KUKA KRL program: MyProgram_254().src

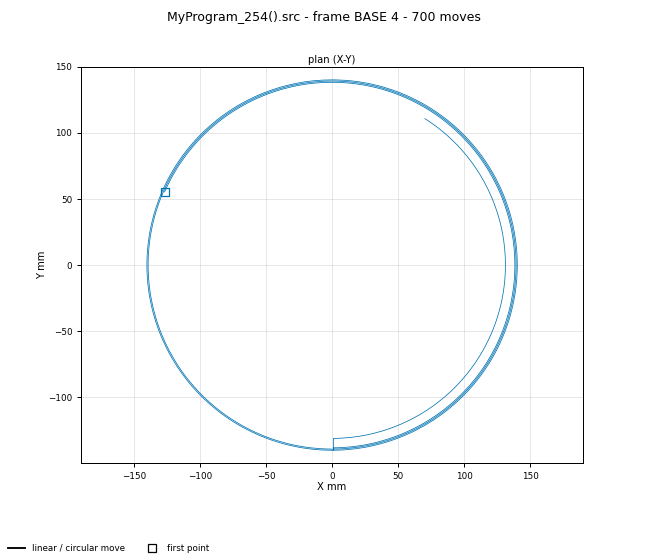
[picture p0: tool path of MyProgram_254().src in frame BASE 4, 700 of 700 moves have a stored position in this frame; points joined in program order, loops and branches not executed]
&ACCESS RVP
&REL 1
&PARAM TEMPLATE = C:\KRC\Roboter\Template\vorgabe
&PARAM EDITMASK = *
DEF MyProgram_254()
; ---- Setting reference (Base) ----
$BASE = BASE_DATA[4]

; --------------------------
; ---- Setting tool (TCP) ----
$TOOL = TOOL_DATA[3]
; --------------------------

$VEL.CP = VEL_APROX_PRINT
Startdeposition()
$VEL.CP = VEL_PRINT
LIN {X -126.8422,Y 55.3756,Z 165,A 156.6903,B 11.101,C 0.1194,E1 10.9554,E2 294.2461} C_DIS
LIN {X -125.3357,Y 58.7076,Z 165,A 155.0353,B 11.101,C 0.1183,E1 10.9574,E2 295.9168} C_DIS
LIN {X -122.9078,Y 63.6351,Z 165,A 152.7935,B 11.1012,C 0.1116,E1 10.9602,E2 298.152} C_DIS
LIN {X -120.9486,Y 67.2845,Z 165,A 151.0182,B 11.1012,C 0.1084,E1 10.9626,E2 299.9329} C_DIS
LIN {X -118.7949,Y 71.0176,Z 165,A 149.2267,B 11.1012,C 0.104,E1 10.9651,E2 301.7233} C_DIS
LIN {X -116.5286,Y 74.6779,Z 165,A 147.4087,B 11.1012,C 0.1002,E1 10.9678,E2 303.5437} C_DIS
LIN {X -114.1724,Y 78.2328,Z 165,A 145.6197,B 11.1012,C 0.0964,E1 10.9706,E2 305.3336} C_DIS
LIN {X -111.5833,Y 81.8833,Z 165,A 143.8556,B 11.1013,C 0.09,E1 10.9735,E2 307.0847} C_DIS
LIN {X -109.7676,Y 84.302,Z 165,A 142.464,B 11.1013,C 0.09,E1 10.9758,E2 308.4922} C_DIS
LIN {X -105.8245,Y 89.2018,Z 165,A 140.1446,B 11.1014,C 0.0779,E1 10.9799,E2 310.7737} C_DIS
LIN {X -101.7242,Y 93.8506,Z 165,A 137.4637,B 11.1014,C 0.0747,E1 10.9849,E2 313.4662} C_DIS
LIN {X -99.2596,Y 96.4535,Z 165,A 135.6559,B 11.1014,C 0.0784,E1 10.9884,E2 315.3122} C_DIS
LIN {X -95.5367,Y 100.1422,Z 165,A 133.2254,B 11.1014,C 0.0795,E1 10.9934,E2 317.7722} C_DIS
LIN {X -92.5514,Y 102.9078,Z 165,A 132.0249,B 11.1015,C 0.0656,E1 10.9957,E2 318.9118} C_DIS
LIN {X -89.9598,Y 105.1813,Z 165,A 130.463,B 11.1015,C 0.0658,E1 10.999,E2 320.4888} C_DIS
LIN {X -85.7237,Y 108.6608,Z 165,A 127.6711,B 11.1015,C 0.0728,E1 11.0053,E2 323.3422} C_DIS
LIN {X -81.9756,Y 111.5155,Z 165,A 126.1993,B 11.1015,C 0.0589,E1 11.0084,E2 324.7536} C_DIS
LIN {X -78.515,Y 113.9787,Z 165,A 124.1886,B 11.1015,C 0.0614,E1 11.0131,E2 326.7935} C_DIS
LIN {X -75.7163,Y 115.8572,Z 165,A 122.4523,B 11.1015,C 0.0665,E1 11.0172,E2 328.57} C_DIS
LIN {X -71.399,Y 118.5662,Z 165,A 121.0445,B 11.1016,C 0.0478,E1 11.0204,E2 329.8902} C_DIS
LIN {X -68.2441,Y 120.4101,Z 165,A 119.2823,B 11.1016,C 0.051,E1 11.0247,E2 331.6816} C_DIS
LIN {X -63.7093,Y 122.8686,Z 165,A 117.2886,B 11.1016,C 0.0448,E1 11.0296,E2 333.656} C_DIS
LIN {X -60.9978,Y 124.2356,Z 165,A 116.0089,B 11.1016,C 0.0436,E1 11.0328,E2 334.9372} C_DIS
LIN {X -57.5207,Y 125.8845,Z 165,A 114.3137,B 11.1016,C 0.0438,E1 11.0371,E2 336.6437} C_DIS
LIN {X -51.8029,Y 128.3418,Z 165,A 112.121,B 11.1016,C 0.0321,E1 11.0426,E2 338.7871} C_DIS
LIN {X -47.623,Y 129.9529,Z 165,A 109.8531,B 11.1016,C 0.0394,E1 11.0487,E2 341.1045} C_DIS
LIN {X -41.2518,Y 132.1139,Z 165,A 107.1931,B 11.1016,C 0.0339,E1 11.0557,E2 343.7469} C_DIS
LIN {X -37.1736,Y 133.3167,Z 165,A 105.423,B 11.1016,C 0.0326,E1 11.0604,E2 345.517} C_DIS
LIN {X -33.4821,Y 134.2926,Z 165,A 103.8309,B 11.1016,C 0.0316,E1 11.0647,E2 347.1094} C_DIS
LIN {X -30.6402,Y 134.9682,Z 165,A 102.5955,B 11.1016,C 0.0314,E1 11.0681,E2 348.3471} C_DIS
LIN {X -27.1287,Y 135.7184,Z 165,A 101.1183,B 11.1016,C 0.0302,E1 11.0721,E2 349.8223} C_DIS
LIN {X -23.4156,Y 136.4088,Z 165,A 99.4566,B 11.1016,C 0.0316,E1 11.0767,E2 351.495} C_DIS
LIN {X -17.5124,Y 137.2909,Z 165,A 96.6135,B 11.1016,C 0.0391,E1 11.0847,E2 354.3821} C_DIS
LIN {X -13.432,Y 137.7494,Z 165,A 95.3157,B 11.1016,C 0.0291,E1 11.0882,E2 355.6298} C_DIS
LIN {X -9.8216,Y 138.0539,Z 165,A 93.3256,B 11.1016,C 0.0402,E1 11.0939,E2 357.679} C_DIS
LIN {X -5.232,Y 138.3038,Z 165,A 91.9382,B 11.1016,C 0.0278,E1 11.0976,E2 359.0024} C_DIS
LIN {X 1.2558,Y 138.3979,Z 165,A 89.3357,B 11.1016,C 0.0256,E1 11.1048,E2 361.5934} C_DIS
LIN {X 4.3034,Y 138.3365,Z 165,A 87.9255,B 11.1016,C 0.0292,E1 11.1088,E2 363.0213} C_DIS
LIN {X 8.1597,Y 138.1623,Z 165,A 86.3703,B 11.1016,C 0.0283,E1 11.1131,E2 364.5706} C_DIS
LIN {X 14.259,Y 137.6672,Z 165,A 83.9892,B 11.1016,C 0.0252,E1 11.1197,E2 366.932} C_DIS
LIN {X 17.7493,Y 137.2599,Z 165,A 81.4648,B 11.1016,C 0.0513,E1 11.1271,E2 369.5867} C_DIS
LIN {X 24.5882,Y 136.201,Z 165,A 79.5411,B 11.1016,C 0.0299,E1 11.132,E2 371.3948} C_DIS
LIN {X 27.7601,Y 135.59,Z 165,A 78.239,B 11.1016,C 0.0298,E1 11.1356,E2 372.6922} C_DIS
LIN {X 30.9188,Y 134.9046,Z 165,A 76.9268,B 11.1016,C 0.0299,E1 11.1391,E2 374.0009} C_DIS
LIN {X 34.1102,Y 134.1332,Z 165,A 75.4988,B 11.1016,C 0.0325,E1 11.143,E2 375.4372} C_DIS
LIN {X 38.047,Y 133.0724,Z 165,A 73.6842,B 11.1016,C 0.0369,E1 11.148,E2 377.2672} C_DIS
LIN {X 41.9679,Y 131.8859,Z 165,A 72.156,B 11.1016,C 0.0341,E1 11.152,E2 378.7744} C_DIS
LIN {X 45.8982,Y 130.5714,Z 165,A 70.4518,B 11.1016,C 0.0354,E1 11.1565,E2 380.4771} C_DIS
LIN {X 49.5024,Y 129.2485,Z 165,A 68.7992,B 11.1016,C 0.0385,E1 11.1608,E2 382.1373} C_DIS
LIN {X 53.1073,Y 127.8078,Z 165,A 66.8551,B 11.1016,C 0.0486,E1 11.166,E2 384.1227} C_DIS
LIN {X 56.8116,Y 126.205,Z 165,A 65.6083,B 11.1016,C 0.04,E1 11.169,E2 385.3173} C_DIS
LIN {X 59.8917,Y 124.7726,Z 165,A 64.1958,B 11.1016,C 0.0418,E1 11.1726,E2 386.7307} C_DIS
LIN {X 63.133,Y 123.1646,Z 165,A 62.7246,B 11.1016,C 0.043,E1 11.1762,E2 388.1986} C_DIS
LIN {X 66.3531,Y 121.4618,Z 165,A 61.1606,B 11.1016,C 0.0465,E1 11.1801,E2 389.7697} C_DIS
LIN {X 70.2836,Y 119.2307,Z 165,A 59.3163,B 11.1016,C 0.0485,E1 11.1845,E2 391.6109} C_DIS
LIN {X 74.0781,Y 116.911,Z 165,A 57.4446,B 11.1016,C 0.052,E1 11.189,E2 393.4867} C_DIS
LIN {X 77.9215,Y 114.3858,Z 165,A 55.5169,B 11.1016,C 0.0557,E1 11.1935,E2 395.4177} C_DIS
LIN {X 81.8053,Y 111.6405,Z 165,A 53.5906,B 11.1016,C 0.0579,E1 11.1978,E2 397.3392} C_DIS
LIN {X 85.2293,Y 109.0494,Z 165,A 51.8672,B 11.1016,C 0.0596,E1 11.2016,E2 399.0564} C_DIS
LIN {X 89.6016,Y 105.4858,Z 165,A 49.5456,B 11.1016,C 0.0635,E1 11.2066,E2 401.377} C_DIS
LIN {X 92.8954,Y 102.5971,Z 165,A 47.7257,B 11.1016,C 0.0671,E1 11.2104,E2 403.1982} C_DIS
LIN {X 97.619,Y 98.1134,Z 165,A 43.8812,B 11.1012,C 0.1022,E1 11.2184,E2 407.1848} C_DIS
LIN {X 103.571,Y 91.8083,Z 165,A 41.7812,B 11.1015,C 0.0711,E1 11.222,E2 409.103} C_DIS
LIN {X 105.6642,Y 89.3917,Z 165,A 40.2086,B 11.1015,C 0.0806,E1 11.2249,E2 410.7073} C_DIS
LIN {X 108.4169,Y 86.032,Z 165,A 38.4233,B 11.1014,C 0.0843,E1 11.228,E2 412.492} C_DIS
LIN {X 111.2183,Y 82.379,Z 165,A 36.5371,B 11.1014,C 0.0882,E1 11.2312,E2 414.3767} C_DIS
LIN {X 113.8496,Y 78.7029,Z 165,A 34.6388,B 11.1014,C 0.0933,E1 11.2342,E2 416.2795} C_DIS
LIN {X 116.3557,Y 74.948,Z 165,A 32.7915,B 11.1013,C 0.0973,E1 11.2371,E2 418.1253} C_DIS
LIN {X 118.8953,Y 70.8491,Z 165,A 30.8267,B 11.1013,C 0.1014,E1 11.2399,E2 420.0874} C_DIS
LIN {X 121.4189,Y 66.4319,Z 165,A 29.1082,B 11.1013,C 0.0963,E1 11.2422,E2 421.7587} C_DIS
LIN {X 122.674,Y 64.0805,Z 165,A 27.7823,B 11.1013,C 0.1051,E1 11.244,E2 423.1133} C_DIS
LIN {X 124.1457,Y 61.18,Z 165,A 26.3541,B 11.1012,C 0.1108,E1 11.2458,E2 424.5526} C_DIS
LIN {X 125.7601,Y 57.7898,Z 165,A 24.9307,B 11.1012,C 0.1114,E1 11.2474,E2 425.9608} C_DIS
LIN {X 127.1163,Y 54.7417,Z 165,A 23.3724,B 11.1011,C 0.1198,E1 11.2492,E2 427.5424} C_DIS
LIN {X 128.7891,Y 50.684,Z 165,A 21.4047,B 11.101,C 0.1288,E1 11.2513,E2 429.5304} C_DIS
LIN {X 130.0514,Y 47.3496,Z 165,A 20.4438,B 11.101,C 0.1189,E1 11.2521,E2 430.4279} C_DIS
LIN {X 130.8432,Y 45.1143,Z 165,A 19.2704,B 11.101,C 0.1268,E1 11.2532,E2 431.6262} C_DIS
LIN {X 132.2368,Y 40.8504,Z 165,A 17.4367,B 11.101,C 0.1313,E1 11.2548,E2 433.4586} C_DIS
LIN {X 133.2658,Y 37.3557,Z 165,A 15.9882,B 11.101,C 0.1339,E1 11.2559,E2 434.9009} C_DIS
LIN {X 134.2147,Y 33.7892,Z 165,A 14.5205,B 11.1009,C 0.1366,E1 11.2569,E2 436.3624} C_DIS
LIN {X 135.0364,Y 30.3417,Z 165,A 13.0331,B 11.1009,C 0.1414,E1 11.2579,E2 437.8536} C_DIS
LIN {X 135.8076,Y 26.6838,Z 165,A 11.5685,B 11.1008,C 0.1435,E1 11.2587,E2 439.3092} C_DIS
LIN {X 136.463,Y 23.0912,Z 165,A 9.5984,B 11.1006,C 0.1604,E1 11.2597,E2 441.3383} C_DIS
LIN {X 137.0881,Y 19.0373,Z 165,A 8.566,B 11.1007,C 0.1471,E1 11.2601,E2 442.2886} C_DIS
LIN {X 137.7959,Y 12.9471,Z 165,A 5.7969,B 11.1006,C 0.1609,E1 11.2609,E2 445.0895} C_DIS
LIN {X 138.283,Y 5.7656,Z 165,A 2.9781,B 11.1005,C 0.1652,E1 11.2614,E2 447.891} C_DIS
LIN {X 138.4042,Y 0.3906,Z 165,A 0.8598,B 11.1005,C 0.1688,E1 11.2615,E2 449.9981} C_DIS
LIN {X 138.3759,Y -2.7624,Z 165,A -0.7081,B 11.1003,C 0.1799,E1 11.2615,E2 451.6006} C_DIS
LIN {X 138.2335,Y -6.8405,Z 165,A -2.5356,B 11.1001,C 0.1886,E1 11.2612,E2 453.4472} C_DIS
LIN {X 138.0319,Y -10.1234,Z 165,A -4.1847,B 11.0999,C 0.2004,E1 11.2609,E2 455.1339} C_DIS
LIN {X 137.5769,Y -15.0977,Z 165,A -5.6088,B 11.1001,C 0.1889,E1 11.2605,E2 456.4791} C_DIS
LIN {X 137.1527,Y -18.5674,Z 165,A -7.3816,B 11.0999,C 0.2021,E1 11.2598,E2 458.2948} C_DIS
LIN {X 136.6347,Y -22.0622,Z 165,A -8.7686,B 11.0999,C 0.2043,E1 11.2592,E2 459.6739} C_DIS
LIN {X 135.5552,Y -27.931,Z 165,A -10.9138,B 11.0999,C 0.2026,E1 11.2581,E2 461.7806} C_DIS
LIN {X 134.7931,Y -31.407,Z 165,A -12.4315,B 11.0998,C 0.2081,E1 11.2572,E2 463.3056} C_DIS
LIN {X 133.8602,Y -35.1697,Z 165,A -14.0414,B 11.0997,C 0.2128,E1 11.256,E2 464.918} C_DIS
LIN {X 132.777,Y -39.0578,Z 165,A -15.6348,B 11.0997,C 0.2155,E1 11.2548,E2 466.5034} C_DIS
LIN {X 131.7684,Y -42.336,Z 165,A -17.0131,B 11.0996,C 0.2184,E1 11.2537,E2 467.8781} C_DIS
LIN {X 130.7542,Y -45.371,Z 165,A -18.3519,B 11.0996,C 0.2225,E1 11.2525,E2 469.2201} C_DIS
LIN {X 128.728,Y -50.8411,Z 165,A -20.7081,B 11.0994,C 0.2276,E1 11.2502,E2 471.5717} C_DIS
LIN {X 127.5338,Y -53.7634,Z 165,A -22.006,B 11.0994,C 0.231,E1 11.2488,E2 472.8699} C_DIS
LIN {X 126.1877,Y -56.8503,Z 165,A -23.4176,B 11.0992,C 0.2353,E1 11.2472,E2 474.2853} C_DIS
LIN {X 124.4786,Y -60.5019,Z 165,A -25.4573,B 11.0989,C 0.2498,E1 11.2446,E2 476.3739} C_DIS
LIN {X 122.6847,Y -64.0602,Z 165,A -26.6913,B 11.0991,C 0.2429,E1 11.2431,E2 477.5571} C_DIS
LIN {X 120.5129,Y -68.0619,Z 165,A -28.6313,B 11.0989,C 0.2494,E1 11.2405,E2 479.5064} C_DIS
LIN {X 118.2007,Y -72.0024,Z 165,A -30.4602,B 11.0989,C 0.2526,E1 11.2379,E2 481.3295} C_DIS
LIN {X 115.8546,Y -75.7205,Z 165,A -32.3269,B 11.0987,C 0.2585,E1 11.235,E2 483.2041} C_DIS
LIN {X 113.2407,Y -79.5757,Z 165,A -34.0728,B 11.0987,C 0.2583,E1 11.2323,E2 484.929} C_DIS
LIN {X 109.6989,Y -84.392,Z 165,A -36.4943,B 11.0987,C 0.2629,E1 11.2283,E2 487.3465} C_DIS
LIN {X 107.4958,Y -87.1808,Z 165,A -38.1297,B 11.0984,C 0.2708,E1 11.2254,E2 489.0045} C_DIS
LIN {X 104.3038,Y -90.9748,Z 165,A -40.3713,B 11.0982,C 0.2806,E1 11.2213,E2 491.2722} C_DIS
LIN {X 101.9397,Y -93.6162,Z 165,A -41.5909,B 11.0982,C 0.2773,E1 11.219,E2 492.462} C_DIS
LIN {X 98.7243,Y -97.0012,Z 165,A -43.4925,B 11.0982,C 0.2807,E1 11.2153,E2 494.3617} C_DIS
LIN {X 95.4442,Y -100.2305,Z 165,A -45.3552,B 11.0982,C 0.2837,E1 11.2116,E2 496.2209} C_DIS
LIN {X 92.1717,Y -103.2479,Z 165,A -47.2015,B 11.098,C 0.2876,E1 11.2078,E2 498.0697} C_DIS
LIN {X 88.6911,Y -106.253,Z 165,A -49.1027,B 11.098,C 0.2913,E1 11.2037,E2 499.9726} C_DIS
LIN {X 85.351,Y -108.9538,Z 165,A -50.85,B 11.0979,C 0.2939,E1 11.1999,E2 501.7177} C_DIS
LIN {X 81.7089,Y -111.7114,Z 165,A -52.7213,B 11.0978,C 0.2969,E1 11.1957,E2 503.5884} C_DIS
LIN {X 78.2131,Y -114.1859,Z 165,A -54.4818,B 11.0978,C 0.2997,E1 11.1917,E2 505.349} C_DIS
LIN {X 74.5541,Y -116.6079,Z 165,A -56.903,B 11.0972,C 0.3186,E1 11.1859,E2 507.8487} C_DIS
LIN {X 69.7904,Y -119.5204,Z 165,A -58.2736,B 11.0978,C 0.2978,E1 11.1828,E2 509.1019} C_DIS
LIN {X 65.5762,Y -121.883,Z 165,A -60.6286,B 11.0974,C 0.3101,E1 11.177,E2 511.5041} C_DIS
LIN {X 61.1994,Y -124.1361,Z 165,A -62.8101,B 11.0972,C 0.3168,E1 11.1715,E2 513.7057} C_DIS
LIN {X 58.1504,Y -125.5933,Z 165,A -63.6094,B 11.0976,C 0.3031,E1 11.1697,E2 514.4295} C_DIS
LIN {X 55.3806,Y -126.84,Z 165,A -65.1912,B 11.0973,C 0.3132,E1 11.1655,E2 516.0541} C_DIS
LIN {X 51.7812,Y -128.3506,Z 165,A -66.7707,B 11.0973,C 0.3143,E1 11.1614,E2 517.6303} C_DIS
LIN {X 47.9975,Y -129.8143,Z 165,A -68.4012,B 11.0973,C 0.315,E1 11.1572,E2 519.2559} C_DIS
LIN {X 44.99,Y -130.8863,Z 165,A -69.7053,B 11.0973,C 0.316,E1 11.1538,E2 520.5588} C_DIS
LIN {X 41.9118,Y -131.9039,Z 165,A -71.0434,B 11.0973,C 0.3173,E1 11.1502,E2 521.8973} C_DIS
LIN {X 38.7235,Y -132.8748,Z 165,A -72.4527,B 11.0972,C 0.3193,E1 11.1464,E2 523.3114} C_DIS
LIN {X 35.4847,Y -133.7762,Z 165,A -73.8521,B 11.0972,C 0.3208,E1 11.1426,E2 524.7128} C_DIS
LIN {X 32.3343,Y -134.5723,Z 165,A -75.1931,B 11.0971,C 0.3218,E1 11.139,E2 526.0542} C_DIS
LIN {X 28.5136,Y -135.435,Z 165,A -77.2887,B 11.0967,C 0.3349,E1 11.1331,E2 528.2114} C_DIS
LIN {X 24.2533,Y -136.2609,Z 165,A -78.6322,B 11.097,C 0.3248,E1 11.1296,E2 529.4984} C_DIS
LIN {X 19.7683,Y -136.9836,Z 165,A -80.9345,B 11.0967,C 0.3364,E1 11.1231,E2 531.8555} C_DIS
LIN {X 15.4099,Y -137.5433,Z 165,A -82.3073,B 11.097,C 0.3261,E1 11.1194,E2 533.1727} C_DIS
LIN {X 9.201,Y -138.0982,Z 165,A -84.7884,B 11.097,C 0.3246,E1 11.1125,E2 535.6426} C_DIS
LIN {X 4.5834,Y -138.3287,Z 165,A -86.8082,B 11.097,C 0.3278,E1 11.1069,E2 537.677} C_DIS
LIN {X 0.9854,Y -138.3876,Z 165,A -87.957,B 11.0972,C 0.3195,E1 11.1038,E2 538.7825} C_DIS
Enddeposition()
LIN {X 0.9854,Y -138.3876,Z 165,A -87.957,B 11.0972,C 0.3195,E1 11.1038,E2 538.7825} C_DIS
Startdeposition()
$VEL.CP = VEL_PRINT
LIN {X 1.7012,Y -139.3118,Z 165,A -87.2529,B 11.0972,C 0.316,E1 11.1058,E2 538.0605} C_DIS
LIN {X 4.8035,Y -139.2394,Z 165,A -86.1094,B 11.0972,C 0.3191,E1 11.1089,E2 536.9335} C_DIS
LIN {X 8.5437,Y -139.0585,Z 165,A -84.6161,B 11.0972,C 0.3198,E1 11.1131,E2 535.4454} C_DIS
LIN {X 11.9095,Y -138.8109,Z 165,A -82.6979,B 11.0976,C 0.3058,E1 11.1186,E2 533.4573} C_DIS
LIN {X 15.9063,Y -138.411,Z 165,A -81.5355,B 11.0972,C 0.3176,E1 11.1217,E2 532.3579} C_DIS
LIN {X 19.0739,Y -138.0103,Z 165,A -80.1038,B 11.0973,C 0.3139,E1 11.1257,E2 530.9099} C_DIS
LIN {X 22.5607,Y -137.4823,Z 165,A -78.7699,B 11.0973,C 0.316,E1 11.1293,E2 529.5902} C_DIS
LIN {X 25.6774,Y -136.9348,Z 165,A -77.4876,B 11.0973,C 0.3156,E1 11.1328,E2 528.3095} C_DIS
LIN {X 31.415,Y -135.733,Z 165,A -74.8742,B 11.0975,C 0.3086,E1 11.1401,E2 525.6682} C_DIS
LIN {X 35.6642,Y -134.6785,Z 165,A -73.1892,B 11.0975,C 0.31,E1 11.1446,E2 523.997} C_DIS
LIN {X 38.9696,Y -133.7594,Z 165,A -71.867,B 11.0975,C 0.311,E1 11.1481,E2 522.6853} C_DIS
LIN {X 41.7152,Y -132.9305,Z 165,A -70.6762,B 11.0975,C 0.3096,E1 11.1513,E2 521.4921} C_DIS
LIN {X 45.2574,Y -131.7653,Z 165,A -69.0738,B 11.0975,C 0.3062,E1 11.1556,E2 519.8795} C_DIS
LIN {X 48.2763,Y -130.6903,Z 165,A -67.8684,B 11.0975,C 0.3076,E1 11.1587,E2 518.6878} C_DIS
LIN {X 50.975,Y -129.661,Z 165,A -66.4976,B 11.0977,C 0.3014,E1 11.1623,E2 517.2921} C_DIS
LIN {X 55.0021,Y -128.0039,Z 165,A -64.8478,B 11.0977,C 0.3029,E1 11.1665,E2 515.6591} C_DIS
LIN {X 58.2988,Y -126.5362,Z 165,A -62.9581,B 11.098,C 0.2901,E1 11.1715,E2 513.7151} C_DIS
LIN {X 61.7984,Y -124.8644,Z 165,A -61.7868,B 11.0977,C 0.2991,E1 11.1743,E2 512.5978} C_DIS
LIN {X 64.8483,Y -123.3078,Z 165,A -60.4263,B 11.0977,C 0.2983,E1 11.1776,E2 511.2423} C_DIS
LIN {X 68.4322,Y -121.358,Z 165,A -58.6045,B 11.0979,C 0.292,E1 11.1821,E2 509.4003} C_DIS
LIN {X 71.297,Y -119.6972,Z 165,A -57.1284,B 11.0981,C 0.2867,E1 11.1857,E2 507.908} C_DIS
LIN {X 75.6284,Y -117.009,Z 165,A -55.1876,B 11.0981,C 0.2874,E1 11.1902,E2 505.9854} C_DIS
LIN {X 79.2835,Y -114.5641,Z 165,A -53.3454,B 11.0981,C 0.2833,E1 11.1945,E2 504.1371} C_DIS
LIN {X 83.1086,Y -111.8198,Z 165,A -51.4645,B 11.0981,C 0.2812,E1 11.1987,E2 502.2614} C_DIS
LIN {X 86.5638,Y -109.1671,Z 165,A -49.6854,B 11.0983,C 0.2781,E1 11.2026,E2 500.4822} C_DIS
LIN {X 89.9951,Y -106.3563,Z 165,A -47.8785,B 11.0983,C 0.275,E1 11.2065,E2 498.6756} C_DIS
LIN {X 93.2139,Y -103.547,Z 165,A -46.1211,B 11.0984,C 0.2714,E1 11.2102,E2 496.9163} C_DIS
LIN {X 96.3807,Y -100.6055,Z 165,A -44.3921,B 11.0984,C 0.269,E1 11.2137,E2 495.1917} C_DIS
LIN {X 99.4864,Y -97.5353,Z 165,A -42.6242,B 11.0986,C 0.2658,E1 11.2172,E2 493.4255} C_DIS
LIN {X 102.4384,Y -94.4304,Z 165,A -40.8125,B 11.0986,C 0.2605,E1 11.2206,E2 491.6054} C_DIS
LIN {X 105.659,Y -90.8123,Z 165,A -38.9253,B 11.0987,C 0.2588,E1 11.2241,E2 489.7297} C_DIS
LIN {X 108.2672,Y -87.6868,Z 165,A -37.2697,B 11.0988,C 0.2554,E1 11.227,E2 488.0747} C_DIS
LIN {X 110.6535,Y -84.6551,Z 165,A -35.6595,B 11.0989,C 0.251,E1 11.2298,E2 486.4596} C_DIS
LIN {X 114.1805,Y -79.8348,Z 165,A -32.5812,B 11.0994,C 0.2277,E1 11.2349,E2 483.2971} C_DIS
LIN {X 117.409,Y -75.0054,Z 165,A -30.5838,B 11.0994,C 0.2325,E1 11.2379,E2 481.3485} C_DIS
LIN {X 119.4291,Y -71.7463,Z 165,A -29.2995,B 11.0992,C 0.2366,E1 11.2397,E2 480.1006} C_DIS
LIN {X 121.659,Y -67.8966,Z 165,A -27.4727,B 11.0993,C 0.2319,E1 11.2422,E2 478.2721} C_DIS
LIN {X 123.635,Y -64.2252,Z 165,A -25.5533,B 11.0995,C 0.2216,E1 11.2447,E2 476.324} C_DIS
LIN {X 125.2984,Y -60.9187,Z 165,A -24.2618,B 11.0995,C 0.224,E1 11.2462,E2 475.0608} C_DIS
LIN {X 127.0205,Y -57.2369,Z 165,A -22.71,B 11.0995,C 0.2227,E1 11.248,E2 473.5226} C_DIS
LIN {X 128.2369,Y -54.4623,Z 165,A -21.3509,B 11.0996,C 0.2162,E1 11.2496,E2 472.1475} C_DIS
LIN {X 129.5719,Y -51.2042,Z 165,A -20.111,B 11.0996,C 0.218,E1 11.2508,E2 470.933} C_DIS
LIN {X 130.4137,Y -49.0147,Z 165,A -19.0482,B 11.0997,C 0.2125,E1 11.2519,E2 469.8562} C_DIS
LIN {X 131.9571,Y -44.6991,Z 165,A -17.2837,B 11.0997,C 0.2106,E1 11.2535,E2 468.1053} C_DIS
LIN {X 133.0155,Y -41.4432,Z 165,A -15.7728,B 11.0999,C 0.2037,E1 11.2548,E2 466.5795} C_DIS
LIN {X 134.2629,Y -37.1991,Z 165,A -14.0285,B 11.0999,C 0.2006,E1 11.2561,E2 464.8428} C_DIS
LIN {X 135.3597,Y -32.9859,Z 165,A -12.2523,B 11.1,C 0.1959,E1 11.2573,E2 463.0664} C_DIS
LIN {X 136.3787,Y -28.4883,Z 165,A -9.9438,B 11.1003,C 0.1788,E1 11.2587,E2 460.7023} C_DIS
LIN {X 137.2137,Y -24.1407,Z 165,A -8.5562,B 11.1002,C 0.1857,E1 11.2594,E2 459.369} C_DIS
LIN {X 137.9303,Y -19.6332,Z 165,A -6.7585,B 11.1002,C 0.1824,E1 11.2601,E2 457.5795} C_DIS
LIN {X 138.4539,Y -15.5298,Z 165,A -5.0383,B 11.1003,C 0.1769,E1 11.2607,E2 455.855} C_DIS
LIN {X 138.8809,Y -11.0799,Z 165,A -3.3233,B 11.1003,C 0.1749,E1 11.2611,E2 454.1539} C_DIS
LIN {X 139.0862,Y -8.0945,Z 165,A -1.9489,B 11.1005,C 0.1673,E1 11.2613,E2 452.7597} C_DIS
LIN {X 139.2563,Y -4.2555,Z 165,A -0.6599,B 11.1005,C 0.1708,E1 11.2615,E2 451.5066} C_DIS
LIN {X 139.321,Y -0.5795,Z 165,A 0.986,B 11.1005,C 0.1626,E1 11.2615,E2 449.8418} C_DIS
LIN {X 139.266,Y 3.9078,Z 165,A 2.8765,B 11.1006,C 0.1559,E1 11.2615,E2 447.9436} C_DIS
LIN {X 139.0389,Y 8.8631,Z 165,A 4.8544,B 11.1006,C 0.1517,E1 11.2611,E2 445.9718} C_DIS
LIN {X 138.6013,Y 14.1569,Z 165,A 7.1977,B 11.1008,C 0.1409,E1 11.2605,E2 443.6058} C_DIS
LIN {X 137.8694,Y 20.0595,Z 165,A 9.95,B 11.101,C 0.1252,E1 11.2594,E2 440.8115} C_DIS
LIN {X 137.0651,Y 24.9716,Z 165,A 11.3299,B 11.1009,C 0.1379,E1 11.2588,E2 439.5158} C_DIS
LIN {X 135.9456,Y 30.4846,Z 165,A 13.7503,B 11.1009,C 0.1283,E1 11.2574,E2 437.0797} C_DIS
LIN {X 135.1653,Y 33.7757,Z 165,A 14.977,B 11.1009,C 0.1289,E1 11.2566,E2 435.8727} C_DIS
LIN {X 134.2964,Y 37.0793,Z 165,A 16.4828,B 11.101,C 0.1222,E1 11.2555,E2 434.3528} C_DIS
LIN {X 133.4459,Y 40.037,Z 165,A 17.7609,B 11.101,C 0.1183,E1 11.2545,E2 433.0721} C_DIS
LIN {X 132.1774,Y 44.0375,Z 165,A 19.3441,B 11.101,C 0.1175,E1 11.2531,E2 431.5056} C_DIS
LIN {X 131.2468,Y 46.7411,Z 165,A 20.4341,B 11.1011,C 0.1166,E1 11.2521,E2 430.4256} C_DIS
LIN {X 129.7133,Y 50.8405,Z 165,A 23.097,B 11.1014,C 0.0878,E1 11.2493,E2 427.6502} C_DIS
LIN {X 127.3886,Y 56.4141,Z 165,A 24.8058,B 11.1012,C 0.1026,E1 11.2475,E2 426.0395} C_DIS
LIN {X 125.2784,Y 60.9591,Z 165,A 26.9107,B 11.1013,C 0.096,E1 11.245,E2 423.9274} C_DIS
LIN {X 123.5781,Y 64.3336,Z 165,A 28.4011,B 11.1013,C 0.0937,E1 11.2431,E2 422.444} C_DIS
LIN {X 122.1279,Y 67.0492,Z 165,A 29.8901,B 11.1013,C 0.0844,E1 11.2411,E2 420.9257} C_DIS
LIN {X 120.5107,Y 69.9133,Z 165,A 31.3669,B 11.1014,C 0.0776,E1 11.239,E2 419.4321} C_DIS
LIN {X 118.4016,Y 73.4285,Z 165,A 32.7111,B 11.1014,C 0.0828,E1 11.2371,E2 418.1305} C_DIS
LIN {X 116.0954,Y 77.024,Z 165,A 34.4674,B 11.1014,C 0.0786,E1 11.2344,E2 416.3732} C_DIS
LIN {X 113.4442,Y 80.8773,Z 165,A 36.3137,B 11.1014,C 0.0761,E1 11.2314,E2 414.5357} C_DIS
LIN {X 110.9958,Y 84.2065,Z 165,A 37.9978,B 11.1014,C 0.0726,E1 11.2286,E2 412.8527} C_DIS
LIN {X 108.2277,Y 87.7358,Z 165,A 39.7857,B 11.1014,C 0.07,E1 11.2255,E2 411.071} C_DIS
LIN {X 105.4617,Y 91.0414,Z 165,A 41.5124,B 11.1015,C 0.0673,E1 11.2224,E2 409.3492} C_DIS
LIN {X 101.6373,Y 95.2928,Z 165,A 43.8968,B 11.1015,C 0.0614,E1 11.2179,E2 406.9597} C_DIS
LIN {X 98.6648,Y 98.3666,Z 165,A 45.6725,B 11.1015,C 0.0573,E1 11.2144,E2 405.1811} C_DIS
LIN {X 94.9904,Y 101.9191,Z 165,A 47.7613,B 11.1015,C 0.0535,E1 11.2102,E2 403.0932} C_DIS
LIN {X 91.5303,Y 105.0376,Z 165,A 49.5441,B 11.1015,C 0.0535,E1 11.2065,E2 401.3265} C_DIS
LIN {X 88.3475,Y 107.7286,Z 165,A 51.3243,B 11.1016,C 0.0485,E1 11.2027,E2 399.5374} C_DIS
LIN {X 85.1624,Y 110.2638,Z 165,A 52.9542,B 11.1016,C 0.0467,E1 11.1991,E2 397.9127} C_DIS
LIN {X 81.9591,Y 112.6652,Z 165,A 54.6121,B 11.1016,C 0.0436,E1 11.1954,E2 396.253} C_DIS
LIN {X 78.6471,Y 115.0016,Z 165,A 56.2886,B 11.1016,C 0.0406,E1 11.1915,E2 394.5749} C_DIS
LIN {X 74.8275,Y 117.5229,Z 165,A 58.101,B 11.1016,C 0.0395,E1 11.1873,E2 392.771} C_DIS
LIN {X 71.3609,Y 119.6591,Z 165,A 59.8122,B 11.1016,C 0.0361,E1 11.1832,E2 391.0549} C_DIS
LIN {X 67.4293,Y 121.9179,Z 165,A 61.632,B 11.1016,C 0.0347,E1 11.1788,E2 389.2406} C_DIS
LIN {X 63.7863,Y 123.8623,Z 165,A 63.377,B 11.1016,C 0.0312,E1 11.1745,E2 387.4896} C_DIS
LIN {X 60.2297,Y 125.6286,Z 165,A 64.8612,B 11.1016,C 0.033,E1 11.1708,E2 386.0241} C_DIS
LIN {X 57.471,Y 126.9158,Z 165,A 66.2083,B 11.1016,C 0.0291,E1 11.1673,E2 384.665} C_DIS
LIN {X 54.5616,Y 128.1944,Z 165,A 67.4468,B 11.1016,C 0.0294,E1 11.1642,E2 383.4353} C_DIS
LIN {X 52.0776,Y 129.221,Z 165,A 68.4886,B 11.1016,C 0.0299,E1 11.1615,E2 382.4013} C_DIS
LIN {X 48.9187,Y 130.4497,Z 165,A 69.9831,B 11.1016,C 0.0259,E1 11.1576,E2 380.8943} C_DIS
LIN {X 44.9593,Y 131.8686,Z 165,A 71.7653,B 11.1016,C 0.023,E1 11.1529,E2 379.1057} C_DIS
LIN {X 41.2584,Y 133.0721,Z 165,A 73.1883,B 11.1016,C 0.0261,E1 11.1491,E2 377.7052} C_DIS
LIN {X 38.3784,Y 133.9325,Z 165,A 74.5931,B 11.1016,C 0.0209,E1 11.1453,E2 376.2795} C_DIS
LIN {X 33.8756,Y 135.1399,Z 165,A 76.3775,B 11.1016,C 0.0229,E1 11.1405,E2 374.5121} C_DIS
LIN {X 30.0587,Y 136.0409,Z 165,A 78.1049,B 11.1016,C 0.0191,E1 11.1358,E2 372.7707} C_DIS
LIN {X 22.5712,Y 137.4805,Z 165,A 81.1501,B 11.1016,C 0.0199,E1 11.1275,E2 369.7378} C_DIS
LIN {X 18.7194,Y 138.0587,Z 165,A 82.7074,B 11.1016,C 0.0204,E1 11.1232,E2 368.1866} C_DIS
LIN {X 14.8637,Y 138.5255,Z 165,A 84.5576,B 11.1017,C 0.0137,E1 11.118,E2 366.3051} C_DIS
LIN {X 9.5075,Y 138.9974,Z 165,A 86.5624,B 11.1017,C 0.0184,E1 11.1124,E2 364.3272} C_DIS
LIN {X 5.3498,Y 139.2181,Z 165,A 88.3496,B 11.1017,C 0.0164,E1 11.1074,E2 362.5312} C_DIS
LIN {X 0.6797,Y 139.3192,Z 165,A 90.2313,B 11.1017,C 0.0174,E1 11.1022,E2 360.6553} C_DIS
LIN {X -4.5151,Y 139.2491,Z 165,A 92.4365,B 11.1017,C 0.0159,E1 11.096,E2 358.4426} C_DIS
LIN {X -7.8862,Y 139.099,Z 165,A 93.8213,B 11.1017,C 0.0163,E1 11.0922,E2 357.0588} C_DIS
LIN {X -12.652,Y 138.7466,Z 165,A 96.1517,B 11.1017,C 0.0081,E1 11.0856,E2 354.6835} C_DIS
LIN {X -16.9407,Y 138.2876,Z 165,A 97.4027,B 11.1017,C 0.0213,E1 11.0823,E2 353.4993} C_DIS
LIN {X -19.7844,Y 137.9087,Z 165,A 98.949,B 11.1017,C 0.0131,E1 11.0779,E2 351.9077} C_DIS
LIN {X -23.2545,Y 137.3665,Z 165,A 100.1665,B 11.1017,C 0.0193,E1 11.0746,E2 350.7197} C_DIS
LIN {X -26.7982,Y 136.7205,Z 165,A 101.5414,B 11.1017,C 0.0227,E1 11.0709,E2 349.3591} C_DIS
LIN {X -29.8415,Y 136.0878,Z 165,A 102.9588,B 11.1017,C 0.0203,E1 11.067,E2 347.9252} C_DIS
LIN {X -34.1052,Y 135.0817,Z 165,A 104.5936,B 11.1017,C 0.0255,E1 11.0626,E2 346.3125} C_DIS
LIN {X -37.3888,Y 134.2098,Z 165,A 106.0796,B 11.1017,C 0.0246,E1 11.0585,E2 344.8164} C_DIS
LIN {X -40.6306,Y 133.2642,Z 165,A 107.5732,B 11.1017,C 0.0234,E1 11.0545,E2 343.3106} C_DIS
LIN {X -45.4584,Y 131.6956,Z 165,A 109.4126,B 11.1017,C 0.0312,E1 11.0497,E2 341.504} C_DIS
LIN {X -48.8274,Y 130.4839,Z 165,A 110.8688,B 11.1017,C 0.0331,E1 11.0459,E2 340.0509} C_DIS
LIN {X -51.0902,Y 129.6163,Z 165,A 112.1811,B 11.1017,C 0.027,E1 11.0424,E2 338.7} C_DIS
LIN {X -54.3195,Y 128.2965,Z 165,A 113.5864,B 11.1017,C 0.0294,E1 11.0388,E2 337.2995} C_DIS
LIN {X -57.814,Y 126.7604,Z 165,A 115.1382,B 11.1017,C 0.0317,E1 11.0349,E2 335.7513} C_DIS
LIN {X -61.232,Y 125.1438,Z 165,A 117.0167,B 11.1017,C 0.0264,E1 11.03,E2 333.8334} C_DIS
LIN {X -64.6882,Y 123.3919,Z 165,A 118.1593,B 11.1017,C 0.0389,E1 11.0274,E2 332.7489} C_DIS
LIN {X -68.5009,Y 121.3189,Z 165,A 120.1422,B 11.1017,C 0.0371,E1 11.0224,E2 330.7428} C_DIS
LIN {X -71.4315,Y 119.6171,Z 165,A 121.6588,B 11.1017,C 0.0364,E1 11.0188,E2 329.2121} C_DIS
LIN {X -76.0513,Y 116.7345,Z 165,A 123.7563,B 11.1017,C 0.0433,E1 11.0139,E2 327.1347} C_DIS
LIN {X -79.7004,Y 114.274,Z 165,A 125.5451,B 11.1017,C 0.0469,E1 11.0098,E2 325.3502} C_DIS
LIN {X -83.1361,Y 111.7993,Z 165,A 127.4359,B 11.1017,C 0.0466,E1 11.0055,E2 323.4423} C_DIS
LIN {X -87.1447,Y 108.7044,Z 165,A 129.3996,B 11.1016,C 0.0531,E1 11.0012,E2 321.4957} C_DIS
LIN {X -90.505,Y 105.9229,Z 165,A 131.1868,B 11.1016,C 0.0568,E1 10.9974,E2 319.7111} C_DIS
LIN {X -93.6656,Y 103.138,Z 165,A 132.9645,B 11.1016,C 0.0592,E1 10.9937,E2 317.9295} C_DIS
LIN {X -97.236,Y 99.7799,Z 165,A 135.0897,B 11.1016,C 0.061,E1 10.9894,E2 315.7928} C_DIS
LIN {X -100.2049,Y 96.7971,Z 165,A 136.7776,B 11.1016,C 0.0656,E1 10.9861,E2 314.1121} C_DIS
LIN {X -102.819,Y 94.0163,Z 165,A 138.5381,B 11.1016,C 0.0649,E1 10.9827,E2 312.3292} C_DIS
LIN {X -106.8232,Y 89.4399,Z 165,A 141.4209,B 11.1016,C 0.0622,E1 10.9774,E2 309.4008} C_DIS
LIN {X -109.9911,Y 85.5142,Z 165,A 142.8433,B 11.1014,C 0.0813,E1 10.9751,E2 308.063} C_DIS
LIN {X -113.1493,Y 81.2898,Z 165,A 145.2279,B 11.1014,C 0.0819,E1 10.9711,E2 305.6539} C_DIS
LIN {X -115.8869,Y 77.3363,Z 165,A 147.1924,B 11.1014,C 0.087,E1 10.968,E2 303.6932} C_DIS
LIN {X -118.3987,Y 73.4335,Z 165,A 149.0767,B 11.1014,C 0.0924,E1 10.9652,E2 301.8141} C_DIS
LIN {X -120.5497,Y 69.8459,Z 165,A 150.832,B 11.1014,C 0.096,E1 10.9627,E2 300.0564} C_DIS
LIN {X -122.5918,Y 66.1968,Z 165,A 152.6189,B 11.1013,C 0.0991,E1 10.9603,E2 298.263} C_DIS
LIN {X -124.2846,Y 62.9566,Z 165,A 154.1609,B 11.1013,C 0.1022,E1 10.9584,E2 296.7177} C_DIS
LIN {X -126.2911,Y 58.829,Z 165,A 155.7718,B 11.1011,C 0.1132,E1 10.9565,E2 295.1438} C_DIS
LIN {X -127.6565,Y 55.8058,Z 165,A 157.352,B 11.1011,C 0.1123,E1 10.9546,E2 293.538} C_DIS
LIN {X -128.7914,Y 53.1346,Z 165,A 158.8349,B 11.1011,C 0.1094,E1 10.953,E2 292.0199} C_DIS
LIN {X -130.0073,Y 50.0843,Z 165,A 160.023,B 11.1011,C 0.1166,E1 10.9518,E2 290.8539} C_DIS
LIN {X -131.4447,Y 46.182,Z 165,A 161.765,B 11.1011,C 0.1207,E1 10.9502,E2 289.1099} C_DIS
LIN {X -132.5886,Y 42.7856,Z 165,A 162.963,B 11.101,C 0.1307,E1 10.9492,E2 287.9482} C_DIS
LIN {X -133.3414,Y 40.3783,Z 165,A 164.1743,B 11.101,C 0.1299,E1 10.9482,E2 286.7162} C_DIS
LIN {X -134.4429,Y 36.548,Z 165,A 165.9682,B 11.101,C 0.1313,E1 10.9468,E2 284.9046} C_DIS
LIN {X -135.3436,Y 33.0525,Z 165,A 167.3009,B 11.1009,C 0.1388,E1 10.9459,E2 283.5927} C_DIS
LIN {X -136.0388,Y 30.0684,Z 165,A 168.5894,B 11.1009,C 0.1418,E1 10.9451,E2 282.3021} C_DIS
LIN {X -136.6695,Y 27.0593,Z 165,A 169.887,B 11.1008,C 0.1448,E1 10.9444,E2 281.0017} C_DIS
LIN {X -137.2178,Y 24.1181,Z 165,A 171.1288,B 11.1008,C 0.1481,E1 10.9438,E2 279.7598} C_DIS
LIN {X -137.8398,Y 20.2665,Z 165,A 172.85,B 11.1008,C 0.1503,E1 10.9431,E2 278.0256} C_DIS
LIN {X -138.3151,Y 16.7096,Z 165,A 174.2524,B 11.1006,C 0.1562,E1 10.9426,E2 276.634} C_DIS
LIN {X -138.8978,Y 10.8715,Z 165,A 176.7688,B 11.1006,C 0.1611,E1 10.9419,E2 274.1073} C_DIS
LIN {X -139.192,Y 6.0164,Z 165,A 178.8785,B 11.1006,C 0.1646,E1 10.9416,E2 271.9858} C_DIS
LIN {X -139.2952,Y 2.7003,Z 165,A -179.0793,B 11.1006,C 0.1541,E1 10.9416,E2 269.8585} C_DIS
LIN {X -139.2825,Y -3.3127,Z 165,A -177.4734,B 11.1003,C 0.18,E1 10.9416,E2 268.3658} C_DIS
LIN {X -139.1656,Y -6.5871,Z 165,A -176.0425,B 11.1003,C 0.1821,E1 10.9417,E2 266.9257} C_DIS
LIN {X -138.9598,Y -10.0221,Z 165,A -174.5638,B 11.1002,C 0.1849,E1 10.942,E2 265.4404} C_DIS
LIN {X -138.6119,Y -14.0549,Z 165,A -172.8982,B 11.1002,C 0.1897,E1 10.9424,E2 263.7763} C_DIS
LIN {X -138.2703,Y -17.0857,Z 165,A -171.6237,B 11.1001,C 0.193,E1 10.9429,E2 262.5005} C_DIS
LIN {X -137.8575,Y -20.1427,Z 165,A -170.2204,B 11.1001,C 0.1937,E1 10.9434,E2 261.0812} C_DIS
LIN {X -137.2122,Y -24.1496,Z 165,A -168.5768,B 11.0999,C 0.1991,E1 10.9442,E2 259.4425} C_DIS
LIN {X -136.5247,Y -27.771,Z 165,A -167.1369,B 11.0999,C 0.2051,E1 10.945,E2 258.0136} C_DIS
LIN {X -135.8458,Y -30.9213,Z 165,A -165.8903,B 11.0997,C 0.2105,E1 10.9457,E2 256.7782} C_DIS
LIN {X -135.1147,Y -33.9749,Z 165,A -164.6421,B 11.0997,C 0.2151,E1 10.9465,E2 255.5367} C_DIS
LIN {X -134.0405,Y -37.9942,Z 165,A -162.5589,B 11.0997,C 0.2119,E1 10.9481,E2 253.4076} C_DIS
LIN {X -132.9733,Y -41.5809,Z 165,A -160.9888,B 11.0997,C 0.2155,E1 10.9494,E2 251.835} C_DIS
LIN {X -131.8764,Y -44.937,Z 165,A -159.524,B 11.0996,C 0.2192,E1 10.9507,E2 250.3698} C_DIS
LIN {X -130.698,Y -48.2558,Z 165,A -158.2837,B 11.0994,C 0.2277,E1 10.9518,E2 249.1572} C_DIS
LIN {X -129.277,Y -51.9387,Z 165,A -156.6519,B 11.0994,C 0.2319,E1 10.9535,E2 247.5256} C_DIS
LIN {X -127.9923,Y -55.029,Z 165,A -155.1661,B 11.0993,C 0.2332,E1 10.9551,E2 246.0269} C_DIS
LIN {X -126.7545,Y -57.8268,Z 165,A -153.7934,B 11.0993,C 0.234,E1 10.9567,E2 244.6405} C_DIS
LIN {X -125.2891,Y -60.9375,Z 165,A -152.3669,B 11.0993,C 0.2374,E1 10.9585,E2 243.2136} C_DIS
LIN {X -123.555,Y -64.3777,Z 165,A -150.7742,B 11.0991,C 0.2413,E1 10.9605,E2 241.6208} C_DIS
LIN {X -121.4487,Y -68.2708,Z 165,A -148.9347,B 11.0991,C 0.2455,E1 10.963,E2 239.7802} C_DIS
LIN {X -119.1354,Y -72.2321,Z 165,A -147.0183,B 11.0989,C 0.2495,E1 10.9657,E2 237.8612} C_DIS
LIN {X -117.5819,Y -74.7353,Z 165,A -145.6787,B 11.0989,C 0.2495,E1 10.9677,E2 236.5059} C_DIS
LIN {X -114.6754,Y -79.1223,Z 165,A -143.6557,B 11.0988,C 0.2578,E1 10.9709,E2 234.5024} C_DIS
LIN {X -112.2439,Y -82.5347,Z 165,A -141.9785,B 11.0986,C 0.2628,E1 10.9736,E2 232.832} C_DIS
LIN {X -110.0441,Y -85.4458,Z 165,A -140.3495,B 11.0986,C 0.2634,E1 10.9764,E2 231.1874} C_DIS
LIN {X -107.1275,Y -89.0756,Z 165,A -138.6734,B 11.0984,C 0.2729,E1 10.9793,E2 229.5429} C_DIS
LIN {X -101.6496,Y -95.2796,Z 165,A -134.9315,B 11.0984,C 0.2726,E1 10.9864,E2 225.7594} C_DIS
LIN {X -98.5125,Y -98.5199,Z 165,A -133.0556,B 11.0984,C 0.2758,E1 10.99,E2 223.8815} C_DIS
LIN {X -95.1687,Y -101.7531,Z 165,A -131.1521,B 11.0982,C 0.2797,E1 10.9939,E2 221.98} C_DIS
LIN {X -92.9081,Y -103.8208,Z 165,A -129.8395,B 11.0982,C 0.2809,E1 10.9966,E2 220.661} C_DIS
LIN {X -89.5204,Y -106.7557,Z 165,A -128.1043,B 11.0981,C 0.2867,E1 11.0003,E2 218.9403} C_DIS
LIN {X -86.6412,Y -109.1055,Z 165,A -126.5497,B 11.0981,C 0.2888,E1 11.0037,E2 217.3828} C_DIS
LIN {X -83.2896,Y -111.6849,Z 165,A -124.8291,B 11.0979,C 0.2921,E1 11.0075,E2 215.665} C_DIS
LIN {X -80.3102,Y -113.8462,Z 165,A -123.2582,B 11.0979,C 0.2933,E1 11.0111,E2 214.0871} C_DIS
LIN {X -76.7824,Y -116.2549,Z 165,A -121.4339,B 11.0979,C 0.2944,E1 11.0153,E2 212.2544} C_DIS
LIN {X -72.9245,Y -118.7127,Z 165,A -119.5903,B 11.0978,C 0.298,E1 11.0197,E2 210.4158} C_DIS
LIN {X -69.318,Y -120.8545,Z 165,A -117.8292,B 11.0978,C 0.2995,E1 11.0239,E2 208.6503} C_DIS
LIN {X -65.5827,Y -122.9218,Z 165,A -116.014,B 11.0977,C 0.3004,E1 11.0284,E2 206.8276} C_DIS
LIN {X -61.8489,Y -124.8395,Z 165,A -114.4597,B 11.0975,C 0.3065,E1 11.0322,E2 205.2955} C_DIS
LIN {X -58.3144,Y -126.529,Z 165,A -112.8547,B 11.0975,C 0.3085,E1 11.0363,E2 203.6914} C_DIS
LIN {X -55.0882,Y -127.9667,Z 165,A -111.4012,B 11.0975,C 0.31,E1 11.04,E2 202.2377} C_DIS
LIN {X -52.6858,Y -128.9759,Z 165,A -110.3374,B 11.0975,C 0.3113,E1 11.0427,E2 201.1749} C_DIS
LIN {X -50.1445,Y -129.9839,Z 165,A -109.0602,B 11.0975,C 0.3087,E1 11.0461,E2 199.8778} C_DIS
LIN {X -45.9146,Y -131.5374,Z 165,A -107.3085,B 11.0974,C 0.3127,E1 11.0507,E2 198.139} C_DIS
LIN {X -42.9027,Y -132.5512,Z 165,A -106.0686,B 11.0973,C 0.3154,E1 11.0539,E2 196.9078} C_DIS
LIN {X -34.9534,Y -134.8664,Z 165,A -102.3827,B 11.0974,C 0.311,E1 11.064,E2 193.185} C_DIS
LIN {X -31.0721,Y -135.8114,Z 165,A -100.5842,B 11.0974,C 0.308,E1 11.0689,E2 191.3657} C_DIS
LIN {X -27.7291,Y -136.5332,Z 165,A -99.4632,B 11.0973,C 0.3157,E1 11.0719,E2 190.2817} C_DIS
LIN {X -24.0139,Y -137.2364,Z 165,A -97.8541,B 11.0973,C 0.315,E1 11.0763,E2 188.6651} C_DIS
LIN {X -19.8348,Y -137.9015,Z 165,A -96.1904,B 11.0973,C 0.3174,E1 11.0809,E2 187.0108} C_DIS
LIN {X -15.722,Y -138.4324,Z 165,A -94.3335,B 11.0973,C 0.314,E1 11.0861,E2 185.1336} C_DIS
LIN {X -11.5963,Y -138.8373,Z 165,A -92.8556,B 11.0972,C 0.3199,E1 11.0901,E2 183.6845} C_DIS
LIN {X -8.9265,Y -139.035,Z 165,A -91.8105,B 11.0972,C 0.3214,E1 11.093,E2 182.6462} C_DIS
LIN {X -6.3894,Y -139.1755,Z 165,A -90.6611,B 11.0972,C 0.3188,E1 11.0962,E2 181.4829} C_DIS
LIN {X -3.794,Y -139.2692,Z 165,A -89.5747,B 11.0972,C 0.3183,E1 11.0993,E2 180.3935} C_DIS
LIN {X -0.3839,Y -139.3209,Z 165,A -88.1072,B 11.0972,C 0.3165,E1 11.1034,E2 178.917} C_DIS
LIN {X -0.3839,Y -139.3209,Z 165,A -88.1072,B 11.0972,C 0.3165,E1 11.1034,E2 178.917} C_DIS
Enddeposition()
LIN {X 0.9957,Y -140.2345,Z 165,A -87.8901,B 11.0969,C 0.3319,E1 11.1038,E2 178.7799} C_DIS
Startdeposition()
$VEL.CP = VEL_PRINT
LIN {X -1.7117,Y -140.2299,Z 165,A -89.2777,B 11.0966,C 0.3391,E1 11.0999,E2 180.2047} C_DIS
LIN {X -5.0598,Y -140.1482,Z 165,A -90.6885,B 11.0966,C 0.3402,E1 11.0959,E2 181.6215} C_DIS
LIN {X -8.5951,Y -139.9752,Z 165,A -92.0847,B 11.0966,C 0.3389,E1 11.092,E2 183.0119} C_DIS
LIN {X -12.024,Y -139.7226,Z 165,A -93.4892,B 11.0966,C 0.3388,E1 11.0881,E2 184.417} C_DIS
LIN {X -15.3466,Y -139.397,Z 165,A -94.8652,B 11.0966,C 0.3388,E1 11.0843,E2 185.795} C_DIS
LIN {X -18.8739,Y -138.9644,Z 165,A -96.3138,B 11.0966,C 0.3384,E1 11.0803,E2 187.2437} C_DIS
LIN {X -22.1743,Y -138.4764,Z 165,A -97.7073,B 11.0966,C 0.3387,E1 11.0764,E2 188.6416} C_DIS
LIN {X -25.5634,Y -137.8913,Z 165,A -99.1087,B 11.0966,C 0.3381,E1 11.0726,E2 190.0429} C_DIS
LIN {X -28.9351,Y -137.2228,Z 165,A -100.5133,B 11.0966,C 0.3374,E1 11.0687,E2 191.4479} C_DIS
LIN {X -32.0219,Y -136.5362,Z 165,A -101.8912,B 11.0966,C 0.3388,E1 11.0649,E2 192.8373} C_DIS
LIN {X -35.5501,Y -135.6592,Z 165,A -103.2937,B 11.0967,C 0.3359,E1 11.0612,E2 194.2293} C_DIS
LIN {X -38.9436,Y -134.7237,Z 165,A -104.7387,B 11.0967,C 0.3351,E1 11.0573,E2 195.6755} C_DIS
LIN {X -42.2575,Y -133.7211,Z 165,A -106.1527,B 11.0967,C 0.3341,E1 11.0535,E2 197.0895} C_DIS
LIN {X -45.5214,Y -132.6455,Z 165,A -107.5889,B 11.0968,C 0.3337,E1 11.0497,E2 198.53} C_DIS
LIN {X -48.7682,Y -131.4864,Z 165,A -108.9755,B 11.0968,C 0.3319,E1 11.0461,E2 199.914} C_DIS
LIN {X -51.9774,Y -130.2513,Z 165,A -110.4135,B 11.0968,C 0.3314,E1 11.0423,E2 201.3564} C_DIS
LIN {X -55.1557,Y -128.9378,Z 165,A -111.796,B 11.0969,C 0.3294,E1 11.0388,E2 202.736} C_DIS
LIN {X -58.3923,Y -127.5045,Z 165,A -113.2487,B 11.0969,C 0.328,E1 11.0351,E2 204.1896} C_DIS
LIN {X -61.4573,Y -126.0564,Z 165,A -114.6424,B 11.097,C 0.3266,E1 11.0315,E2 205.5843} C_DIS
LIN {X -64.5893,Y -124.4809,Z 165,A -116.066,B 11.097,C 0.3246,E1 11.028,E2 207.0068} C_DIS
LIN {X -68.2893,Y -122.4912,Z 165,A -117.8279,B 11.0971,C 0.3235,E1 11.0237,E2 208.7745} C_DIS
LIN {X -71.3137,Y -120.7552,Z 165,A -119.2509,B 11.0971,C 0.3215,E1 11.0202,E2 210.197} C_DIS
LIN {X -74.2538,Y -118.9696,Z 165,A -120.6789,B 11.0972,C 0.32,E1 11.0168,E2 211.6278} C_DIS
LIN {X -77.8662,Y -116.6371,Z 165,A -122.4408,B 11.0972,C 0.3175,E1 11.0127,E2 213.39} C_DIS
LIN {X -81.3059,Y -114.2664,Z 165,A -124.2002,B 11.0973,C 0.316,E1 11.0087,E2 215.1559} C_DIS
LIN {X -84.878,Y -111.6389,Z 165,A -126.0782,B 11.0973,C 0.3145,E1 11.0045,E2 217.0419} C_DIS
LIN {X -88.2594,Y -108.9849,Z 165,A -127.7502,B 11.0975,C 0.3095,E1 11.0008,E2 218.7026} C_DIS
LIN {X -90.9433,Y -106.7552,Z 165,A -129.1851,B 11.0975,C 0.3072,E1 10.9978,E2 220.1383} C_DIS
LIN {X -93.9507,Y -104.119,Z 165,A -130.8878,B 11.0976,C 0.3057,E1 10.9942,E2 221.8493} C_DIS
LIN {X -96.6638,Y -101.605,Z 165,A -132.3488,B 11.0977,C 0.3017,E1 10.9912,E2 223.3032} C_DIS
LIN {X -99.1639,Y -99.1669,Z 165,A -133.9282,B 11.0977,C 0.3023,E1 10.988,E2 224.9016} C_DIS
LIN {X -102.1511,Y -96.0862,Z 165,A -135.5755,B 11.0979,C 0.2963,E1 10.9849,E2 226.5346} C_DIS
LIN {X -105.0033,Y -92.9606,Z 165,A -137.3082,B 11.0979,C 0.2928,E1 10.9817,E2 228.267} C_DIS
LIN {X -107.4295,Y -90.1457,Z 165,A -138.9594,B 11.0979,C 0.2924,E1 10.9786,E2 229.9345} C_DIS
LIN {X -110.0263,Y -86.9582,Z 165,A -140.5923,B 11.0981,C 0.2877,E1 10.9758,E2 231.5607} C_DIS
LIN {X -113.1232,Y -82.8886,Z 165,A -142.664,B 11.0982,C 0.2825,E1 10.9723,E2 233.6289} C_DIS
LIN {X -115.1212,Y -80.0903,Z 165,A -144.0732,B 11.0982,C 0.2793,E1 10.9701,E2 235.0378} C_DIS
LIN {X -117.2476,Y -76.9441,Z 165,A -145.7433,B 11.0983,C 0.2783,E1 10.9675,E2 236.7222} C_DIS
LIN {X -119.395,Y -73.5681,Z 165,A -147.3829,B 11.0984,C 0.2744,E1 10.965,E2 238.3614} C_DIS
LIN {X -121.5973,Y -69.8687,Z 165,A -149.074,B 11.0986,C 0.2685,E1 10.9627,E2 240.0426} C_DIS
LIN {X -123.2744,Y -66.8648,Z 165,A -150.6175,B 11.0986,C 0.268,E1 10.9606,E2 241.6028} C_DIS
LIN {X -125.2653,Y -63.054,Z 165,A -152.281,B 11.0987,C 0.2615,E1 10.9585,E2 243.2531} C_DIS
LIN {X -126.7513,Y -60.0096,Z 165,A -153.6797,B 11.0987,C 0.2582,E1 10.9568,E2 244.6527} C_DIS
LIN {X -128.1843,Y -56.8838,Z 165,A -155.0173,B 11.0989,C 0.253,E1 10.9552,E2 245.9806} C_DIS
LIN {X -129.5641,Y -53.6667,Z 165,A -156.5298,B 11.0989,C 0.251,E1 10.9536,E2 247.5025} C_DIS
LIN {X -130.8456,Y -50.4617,Z 165,A -157.9748,B 11.099,C 0.248,E1 10.9521,E2 248.9508} C_DIS
LIN {X -132.0428,Y -47.2401,Z 165,A -159.3838,B 11.0991,C 0.2442,E1 10.9507,E2 250.3592} C_DIS
LIN {X -133.1607,Y -43.9907,Z 165,A -160.8175,B 11.0991,C 0.241,E1 10.9495,E2 251.7955} C_DIS
LIN {X -134.1689,Y -40.8117,Z 165,A -162.197,B 11.0992,C 0.2376,E1 10.9483,E2 253.176} C_DIS
LIN {X -135.129,Y -37.511,Z 165,A -163.6308,B 11.0993,C 0.2343,E1 10.9472,E2 254.6124} C_DIS
LIN {X -135.8757,Y -34.7089,Z 165,A -164.9156,B 11.0993,C 0.2331,E1 10.9463,E2 255.9088} C_DIS
LIN {X -136.7402,Y -31.1289,Z 165,A -166.3953,B 11.0994,C 0.2283,E1 10.9454,E2 257.384} C_DIS
LIN {X -137.5448,Y -27.3618,Z 165,A -167.9094,B 11.0996,C 0.2225,E1 10.9445,E2 258.8891} C_DIS
LIN {X -138.1063,Y -24.3652,Z 165,A -169.2221,B 11.0996,C 0.2204,E1 10.9439,E2 260.2091} C_DIS
LIN {X -138.723,Y -20.5766,Z 165,A -170.7715,B 11.0996,C 0.2155,E1 10.9432,E2 261.7547} C_DIS
LIN {X -139.1732,Y -17.268,Z 165,A -172.2168,B 11.0997,C 0.2132,E1 10.9427,E2 263.2089} C_DIS
LIN {X -139.5638,Y -13.7478,Z 165,A -173.7779,B 11.0997,C 0.2114,E1 10.9422,E2 264.783} C_DIS
LIN {X -139.9751,Y -8.5972,Z 165,A -175.7627,B 11.0999,C 0.2026,E1 10.9418,E2 266.7496} C_DIS
LIN {X -140.1136,Y -5.9464,Z 165,A -176.9372,B 11.0999,C 0.2013,E1 10.9417,E2 267.9345} C_DIS
LIN {X -140.2287,Y -1.7797,Z 165,A -178.5312,B 11.1001,C 0.194,E1 10.9416,E2 269.513} C_DIS
LIN {X -140.2325,Y 1.5499,Z 165,A -179.955,B 11.1001,C 0.1914,E1 10.9416,E2 270.9435} C_DIS
LIN {X -140.1489,Y 5.0401,Z 165,A 178.538,B 11.1001,C 0.1889,E1 10.9417,E2 272.4591} C_DIS
LIN {X -139.9786,Y 8.5401,Z 165,A 177.1328,B 11.1003,C 0.1841,E1 10.9419,E2 273.8594} C_DIS
LIN {X -139.7277,Y 11.9634,Z 165,A 175.7112,B 11.1003,C 0.1804,E1 10.9422,E2 275.2819} C_DIS
LIN {X -139.402,Y 15.3,Z 165,A 174.3066,B 11.1003,C 0.1771,E1 10.9426,E2 276.6894} C_DIS
LIN {X -138.964,Y 18.8772,Z 165,A 172.8257,B 11.1004,C 0.173,E1 10.9432,E2 278.1698} C_DIS
LIN {X -138.4757,Y 22.1791,Z 165,A 171.4122,B 11.1004,C 0.1701,E1 10.9438,E2 279.5882} C_DIS
LIN {X -137.8901,Y 25.5699,Z 165,A 169.9954,B 11.1005,C 0.1662,E1 10.9445,E2 281.0048} C_DIS
LIN {X -137.2207,Y 28.9447,Z 165,A 168.5735,B 11.1005,C 0.1625,E1 10.9453,E2 282.4272} C_DIS
LIN {X -136.4689,Y 32.3023,Z 165,A 167.1229,B 11.1006,C 0.1594,E1 10.9462,E2 283.8819} C_DIS
LIN {X -135.6331,Y 35.648,Z 165,A 165.7253,B 11.1006,C 0.1551,E1 10.9471,E2 285.2764} C_DIS
LIN {X -134.8337,Y 38.5668,Z 165,A 164.3338,B 11.1006,C 0.1549,E1 10.9482,E2 286.6861} C_DIS
LIN {X -133.6914,Y 42.3506,Z 165,A 162.8664,B 11.1008,C 0.1472,E1 10.9494,E2 288.1331} C_DIS
LIN {X -132.6461,Y 45.5197,Z 165,A 161.4292,B 11.1008,C 0.1449,E1 10.9507,E2 289.578} C_DIS
LIN {X -131.4883,Y 48.7634,Z 165,A 160.0342,B 11.1008,C 0.1408,E1 10.952,E2 290.9699} C_DIS
LIN {X -130.2544,Y 51.9698,Z 165,A 158.7441,B 11.101,C 0.1345,E1 10.9533,E2 292.2441} C_DIS
LIN {X -129.2334,Y 54.4587,Z 165,A 157.3641,B 11.101,C 0.1374,E1 10.9548,E2 293.6581} C_DIS
LIN {X -127.8535,Y 57.6234,Z 165,A 156.0656,B 11.101,C 0.1312,E1 10.9563,E2 294.941} C_DIS
LIN {X -126.3651,Y 60.8179,Z 165,A 154.5986,B 11.101,C 0.1279,E1 10.958,E2 296.4097} C_DIS
LIN {X -124.5752,Y 64.4094,Z 165,A 152.9457,B 11.101,C 0.1239,E1 10.9601,E2 298.0625} C_DIS
LIN {X -122.4445,Y 68.373,Z 165,A 151.0942,B 11.1011,C 0.1194,E1 10.9626,E2 299.9136} C_DIS
LIN {X -120.7045,Y 71.4,Z 165,A 149.4974,B 11.1011,C 0.1194,E1 10.9649,E2 301.5301} C_DIS
LIN {X -118.3185,Y 75.2877,Z 165,A 147.6562,B 11.1011,C 0.1142,E1 10.9676,E2 303.3664} C_DIS
LIN {X -116.1257,Y 78.6267,Z 165,A 146.1002,B 11.1012,C 0.1085,E1 10.97,E2 304.9111} C_DIS
LIN {X -113.6899,Y 82.1098,Z 165,A 144.343,B 11.1012,C 0.1047,E1 10.9728,E2 306.669} C_DIS
LIN {X -111.4754,Y 85.0917,Z 165,A 142.7209,B 11.1012,C 0.1033,E1 10.9756,E2 308.3024} C_DIS
LIN {X -108.9922,Y 88.2504,Z 165,A 141.1559,B 11.1013,C 0.0979,E1 10.9783,E2 309.856} C_DIS
LIN {X -106.7679,Y 90.9285,Z 165,A 139.7119,B 11.1013,C 0.0951,E1 10.9809,E2 311.3013} C_DIS
LIN {X -103.9653,Y 94.1201,Z 165,A 137.9654,B 11.1013,C 0.0914,E1 10.9841,E2 313.0472} C_DIS
LIN {X -101.4147,Y 96.8628,Z 165,A 136.3312,B 11.1013,C 0.0904,E1 10.9873,E2 314.6928} C_DIS
LIN {X -98.5594,Y 99.7675,Z 165,A 134.735,B 11.1014,C 0.0853,E1 10.9904,E2 316.2788} C_DIS
LIN {X -96.0841,Y 102.153,Z 165,A 133.3209,B 11.1014,C 0.0827,E1 10.9932,E2 317.6926} C_DIS
LIN {X -93.5398,Y 104.4876,Z 165,A 131.7961,B 11.1014,C 0.0823,E1 10.9964,E2 319.2301} C_DIS
LIN {X -90.333,Y 107.2724,Z 165,A 130.1419,B 11.1014,C 0.0771,E1 10.9999,E2 320.8724} C_DIS
LIN {X -87.6356,Y 109.4874,Z 165,A 128.7143,B 11.1015,C 0.0745,E1 11.003,E2 322.2988} C_DIS
LIN {X -84.9244,Y 111.6034,Z 165,A 127.2926,B 11.1015,C 0.0723,E1 11.0061,E2 323.7212} C_DIS
LIN {X -82.1532,Y 113.6584,Z 165,A 125.8781,B 11.1015,C 0.0699,E1 11.0093,E2 325.1349} C_DIS
LIN {X -79.3431,Y 115.6375,Z 165,A 124.4472,B 11.1015,C 0.068,E1 11.0126,E2 326.5678} C_DIS
LIN {X -75.805,Y 117.9873,Z 165,A 122.6998,B 11.1015,C 0.0654,E1 11.0167,E2 328.3151} C_DIS
LIN {X -72.8454,Y 119.8374,Z 165,A 121.2605,B 11.1015,C 0.0635,E1 11.0201,E2 329.7547} C_DIS
LIN {X -69.1916,Y 121.9836,Z 165,A 119.525,B 11.1015,C 0.0609,E1 11.0243,E2 331.4892} C_DIS
LIN {X -66.195,Y 123.635,Z 165,A 118.0911,B 11.1016,C 0.0597,E1 11.0278,E2 332.9263} C_DIS
LIN {X -63.1135,Y 125.235,Z 165,A 116.6871,B 11.1016,C 0.0574,E1 11.0313,E2 334.3272} C_DIS
LIN {X -60.0073,Y 126.7524,Z 165,A 115.2675,B 11.1016,C 0.0557,E1 11.0349,E2 335.7465} C_DIS
LIN {X -56.8803,Y 128.1858,Z 165,A 113.8662,B 11.1016,C 0.0538,E1 11.0385,E2 337.146} C_DIS
LIN {X -53.6612,Y 129.5664,Z 165,A 112.4279,B 11.1016,C 0.0523,E1 11.0421,E2 338.584} C_DIS
LIN {X -50.4702,Y 130.8423,Z 165,A 111.0067,B 11.1016,C 0.0511,E1 11.0458,E2 340.0063} C_DIS
LIN {X -47.2492,Y 132.0396,Z 165,A 109.6089,B 11.1016,C 0.0495,E1 11.0495,E2 341.4022} C_DIS
LIN {X -43.9994,Y 133.1578,Z 165,A 108.1865,B 11.1016,C 0.0485,E1 11.0533,E2 342.8257} C_DIS
LIN {X -40.8189,Y 134.1667,Z 165,A 106.9106,B 11.1016,C 0.0452,E1 11.0566,E2 344.0897} C_DIS
LIN {X -37.5063,Y 135.1303,Z 165,A 105.3915,B 11.1016,C 0.0466,E1 11.0608,E2 345.6215} C_DIS
LIN {X -34.0766,Y 136.0362,Z 165,A 103.9603,B 11.1016,C 0.045,E1 11.0646,E2 347.0494} C_DIS
LIN {X -30.7297,Y 136.8313,Z 165,A 102.543,B 11.1016,C 0.0443,E1 11.0685,E2 348.4673} C_DIS
LIN {X -27.3639,Y 137.5444,Z 165,A 101.1358,B 11.1016,C 0.0435,E1 11.0723,E2 349.8738} C_DIS
LIN {X -24.6532,Y 138.0547,Z 165,A 99.9455,B 11.1016,C 0.0443,E1 11.0756,E2 351.0712} C_DIS
LIN {X -20.7115,Y 138.7029,Z 165,A 98.3766,B 11.1016,C 0.042,E1 11.0799,E2 352.6313} C_DIS
LIN {X -17.346,Y 139.1638,Z 165,A 96.934,B 11.1016,C 0.0427,E1 11.0839,E2 354.0799} C_DIS
LIN {X -13.8455,Y 139.5544,Z 165,A 95.5318,B 11.1016,C 0.0413,E1 11.0878,E2 355.4767} C_DIS
LIN {X -10.4206,Y 139.8513,Z 165,A 94.191,B 11.1016,C 0.0394,E1 11.0915,E2 356.8087} C_DIS
LIN {X -6.992,Y 140.0645,Z 165,A 92.7222,B 11.1016,C 0.0406,E1 11.0956,E2 358.2849} C_DIS
LIN {X -3.4558,Y 140.197,Z 165,A 91.2889,B 11.1016,C 0.0401,E1 11.0996,E2 359.716} C_DIS
LIN {X -0.1135,Y 140.2405,Z 165,A 89.8773,B 11.1016,C 0.0411,E1 11.1036,E2 361.1328} C_DIS
LIN {X 3.3381,Y 140.2003,Z 165,A 88.5649,B 11.1016,C 0.0388,E1 11.1072,E2 362.4323} C_DIS
LIN {X 6.8734,Y 140.0704,Z 165,A 87.0468,B 11.1016,C 0.0406,E1 11.1115,E2 363.9588} C_DIS
LIN {X 10.2036,Y 139.8672,Z 165,A 85.6738,B 11.1016,C 0.0411,E1 11.1153,E2 365.3325} C_DIS
LIN {X 13.6301,Y 139.5751,Z 165,A 84.3298,B 11.1016,C 0.0399,E1 11.119,E2 366.6684} C_DIS
LIN {X 17.0631,Y 139.1976,Z 165,A 82.8781,B 11.1016,C 0.0413,E1 11.1231,E2 368.1248} C_DIS
LIN {X 20.5696,Y 138.724,Z 165,A 81.4465,B 11.1016,C 0.0415,E1 11.127,E2 369.5541} C_DIS
LIN {X 23.9633,Y 138.1782,Z 165,A 80.0535,B 11.1016,C 0.0418,E1 11.1308,E2 370.9453} C_DIS
LIN {X 27.2461,Y 137.5684,Z 165,A 78.7158,B 11.1016,C 0.0418,E1 11.1345,E2 372.2794} C_DIS
LIN {X 30.6289,Y 136.8544,Z 165,A 77.2549,B 11.1016,C 0.0439,E1 11.1385,E2 373.7459} C_DIS
LIN {X 34.3469,Y 135.9675,Z 165,A 75.5999,B 11.1016,C 0.0472,E1 11.143,E2 375.4123} C_DIS
LIN {X 38.7564,Y 134.7785,Z 165,A 73.7568,B 11.1016,C 0.048,E1 11.148,E2 377.2523} C_DIS
LIN {X 42.3488,Y 133.6919,Z 165,A 72.3426,B 11.1016,C 0.0463,E1 11.1517,E2 378.6513} C_DIS
LIN {X 45.5268,Y 132.6436,Z 165,A 70.9282,B 11.1016,C 0.0487,E1 11.1555,E2 380.0714} C_DIS
LIN {X 48.7654,Y 131.4875,Z 165,A 69.7024,B 11.1016,C 0.0455,E1 11.1586,E2 381.2746} C_DIS
LIN {X 51.9748,Y 130.2523,Z 165,A 68.1319,B 11.1016,C 0.0511,E1 11.1628,E2 382.8659} C_DIS
LIN {X 55.1535,Y 128.9387,Z 165,A 66.7625,B 11.1016,C 0.0517,E1 11.1663,E2 384.2308} C_DIS
LIN {X 57.6062,Y 127.8611,Z 165,A 65.6453,B 11.1016,C 0.0536,E1 11.1691,E2 385.3508} C_DIS
LIN {X 61.4688,Y 126.0507,Z 165,A 63.9436,B 11.1016,C 0.0546,E1 11.1734,E2 387.0474} C_DIS
LIN {X 64.5872,Y 124.482,Z 165,A 62.5521,B 11.1016,C 0.0556,E1 11.1769,E2 388.4346} C_DIS
LIN {X 68.0221,Y 122.6391,Z 165,A 60.8794,B 11.1016,C 0.0598,E1 11.181,E2 390.1175} C_DIS
LIN {X 71.3125,Y 120.7559,Z 165,A 59.3935,B 11.1016,C 0.0604,E1 11.1846,E2 391.5957} C_DIS
LIN {X 74.2528,Y 118.9702,Z 165,A 58.0057,B 11.1016,C 0.062,E1 11.1879,E2 392.9814} C_DIS
LIN {X 77.476,Y 116.8974,Z 165,A 56.3368,B 11.1016,C 0.0672,E1 11.1918,E2 394.6637} C_DIS
LIN {X 80.754,Y 114.6567,Z 165,A 54.7479,B 11.1016,C 0.0689,E1 11.1954,E2 396.2487} C_DIS
LIN {X 84.2306,Y 112.1278,Z 165,A 53.1143,B 11.1016,C 0.0687,E1 11.1991,E2 397.8672} C_DIS
LIN {X 86.9154,Y 110.06,Z 165,A 51.6626,B 11.1016,C 0.0729,E1 11.2023,E2 399.3278} C_DIS
LIN {X 90.2477,Y 107.3439,Z 165,A 49.9711,B 11.1016,C 0.0744,E1 11.2059,E2 401.0117} C_DIS
LIN {X 92.9351,Y 105.0258,Z 165,A 48.4072,B 11.1015,C 0.0802,E1 11.2092,E2 402.5904} C_DIS
LIN {X 96.038,Y 102.1965,Z 165,A 46.8331,B 11.1015,C 0.0798,E1 11.2124,E2 404.1472} C_DIS
LIN {X 98.5192,Y 99.8074,Z 165,A 45.4288,B 11.1015,C 0.0825,E1 11.2152,E2 405.5517} C_DIS
LIN {X 101.4932,Y 96.7807,Z 165,A 43.7115,B 11.1015,C 0.0857,E1 11.2186,E2 407.2677} C_DIS
LIN {X 103.9034,Y 94.1883,Z 165,A 42.23,B 11.1015,C 0.0897,E1 11.2214,E2 408.7543} C_DIS
LIN {X 106.7181,Y 90.987,Z 165,A 40.4928,B 11.1014,C 0.0934,E1 11.2245,E2 410.4919} C_DIS
LIN {X 109.4928,Y 87.6288,Z 165,A 38.8168,B 11.1014,C 0.0946,E1 11.2275,E2 412.1556} C_DIS
LIN {X 111.6092,Y 84.9168,Z 165,A 37.4213,B 11.1014,C 0.0975,E1 11.2299,E2 413.5506} C_DIS
LIN {X 113.688,Y 82.1124,Z 165,A 35.8699,B 11.1013,C 0.1042,E1 11.2324,E2 415.1187} C_DIS
LIN {X 116.0944,Y 78.6731,Z 165,A 34.1997,B 11.1013,C 0.1071,E1 11.2351,E2 416.7841} C_DIS
LIN {X 118.4742,Y 75.0418,Z 165,A 32.5658,B 11.1013,C 0.1076,E1 11.2375,E2 418.4014} C_DIS
LIN {X 120.2699,Y 72.1294,Z 165,A 31.182,B 11.1013,C 0.1107,E1 11.2395,E2 419.7843} C_DIS
LIN {X 121.9753,Y 69.2062,Z 165,A 29.8063,B 11.1012,C 0.114,E1 11.2414,E2 421.1601} C_DIS
LIN {X 123.6571,Y 66.1538,Z 165,A 28.3774,B 11.1012,C 0.1178,E1 11.2434,E2 422.5905} C_DIS
LIN {X 125.2648,Y 63.055,Z 165,A 26.987,B 11.1012,C 0.1205,E1 11.2451,E2 423.9774} C_DIS
LIN {X 126.7512,Y 60.0097,Z 165,A 25.6205,B 11.1011,C 0.1236,E1 11.2468,E2 425.3426} C_DIS
LIN {X 128.1834,Y 56.8856,Z 165,A 24.2314,B 11.1011,C 0.1269,E1 11.2484,E2 426.7308} C_DIS
LIN {X 129.552,Y 53.6957,Z 165,A 22.847,B 11.1011,C 0.1298,E1 11.2499,E2 428.112} C_DIS
LIN {X 130.8257,Y 50.5129,Z 165,A 21.453,B 11.101,C 0.1334,E1 11.2513,E2 429.5063} C_DIS
LIN {X 132.0414,Y 47.244,Z 165,A 20.0581,B 11.101,C 0.1365,E1 11.2526,E2 430.8986} C_DIS
LIN {X 133.1602,Y 43.9921,Z 165,A 18.6593,B 11.1009,C 0.1402,E1 11.2539,E2 432.2978} C_DIS
LIN {X 133.9689,Y 41.4652,Z 165,A 17.4568,B 11.1009,C 0.1465,E1 11.2549,E2 433.5162} C_DIS
LIN {X 135.0472,Y 37.8036,Z 165,A 15.9883,B 11.1008,C 0.1483,E1 11.256,E2 434.9745} C_DIS
LIN {X 136.0366,Y 34.075,Z 165,A 14.5407,B 11.1008,C 0.1492,E1 11.257,E2 436.4071} C_DIS
LIN {X 136.8318,Y 30.7278,Z 165,A 13.1383,B 11.1008,C 0.1532,E1 11.2579,E2 437.8104} C_DIS
LIN {X 137.5466,Y 27.3531,Z 165,A 11.7233,B 11.1007,C 0.1574,E1 11.2587,E2 439.2274} C_DIS
LIN {X 138.1746,Y 23.9835,Z 165,A 10.3463,B 11.1007,C 0.1608,E1 11.2594,E2 440.6028} C_DIS
LIN {X 138.7203,Y 20.5951,Z 165,A 8.9687,B 11.1006,C 0.1641,E1 11.26,E2 441.9785} C_DIS
LIN {X 139.1705,Y 17.2902,Z 165,A 7.5665,B 11.1005,C 0.1692,E1 11.2605,E2 443.3871} C_DIS
LIN {X 139.5113,Y 14.2843,Z 165,A 6.2511,B 11.1004,C 0.175,E1 11.2609,E2 444.7139} C_DIS
LIN {X 139.8161,Y 10.9029,Z 165,A 4.8749,B 11.1004,C 0.1788,E1 11.2612,E2 446.0901} C_DIS
LIN {X 140.0645,Y 6.9918,Z 165,A 3.5371,B 11.1004,C 0.1761,E1 11.2614,E2 447.3958} C_DIS
LIN {X 140.1974,Y 3.4438,Z 165,A 2.0148,B 11.1003,C 0.1824,E1 11.2615,E2 448.9288} C_DIS
LIN {X 140.243,Y -0.0003,Z 165,A 0.5715,B 11.1002,C 0.1876,E1 11.2615,E2 450.3783} C_DIS
LIN {X 140.2003,Y -3.3386,Z 165,A -0.7451,B 11.1002,C 0.1902,E1 11.2615,E2 451.6901} C_DIS
LIN {X 140.0704,Y -6.8749,Z 165,A -2.1594,B 11.1001,C 0.1936,E1 11.2613,E2 453.1019} C_DIS
LIN {X 139.867,Y -10.2055,Z 165,A -3.5151,B 11.1001,C 0.1974,E1 11.2611,E2 454.4581} C_DIS
LIN {X 139.5938,Y -13.4347,Z 165,A -4.8346,B 11.1,C 0.2012,E1 11.2607,E2 455.7784} C_DIS
LIN {X 139.2315,Y -16.7791,Z 165,A -6.1998,B 11.0999,C 0.2049,E1 11.2603,E2 457.1439} C_DIS
LIN {X 138.7237,Y -20.5718,Z 165,A -7.692,B 11.0999,C 0.2075,E1 11.2597,E2 458.6287} C_DIS
LIN {X 138.1777,Y -23.9664,Z 165,A -9.0694,B 11.0998,C 0.2109,E1 11.2591,E2 460.0042} C_DIS
LIN {X 137.5678,Y -27.2491,Z 165,A -10.3917,B 11.0998,C 0.2137,E1 11.2584,E2 461.3226} C_DIS
LIN {X 136.8538,Y -30.6312,Z 165,A -11.8378,B 11.0996,C 0.2187,E1 11.2575,E2 462.7746} C_DIS
LIN {X 136.0355,Y -34.0791,Z 165,A -13.2357,B 11.0996,C 0.2215,E1 11.2566,E2 464.1677} C_DIS
LIN {X 135.3011,Y -36.893,Z 165,A -14.5681,B 11.0994,C 0.2289,E1 11.2556,E2 465.5201} C_DIS
LIN {X 134.2005,Y -40.7087,Z 165,A -15.8822,B 11.0995,C 0.225,E1 11.2546,E2 466.7961} C_DIS
LIN {X 133.1937,Y -43.8915,Z 165,A -17.3834,B 11.0994,C 0.2327,E1 11.2533,E2 468.3167} C_DIS
LIN {X 132.0411,Y -47.2451,Z 165,A -18.713,B 11.0994,C 0.2334,E1 11.2521,E2 469.6325} C_DIS
LIN {X 130.877,Y -50.3811,Z 165,A -20.1597,B 11.0992,C 0.2395,E1 11.2507,E2 471.0912} C_DIS
LIN {X 129.5637,Y -53.6678,Z 165,A -21.5576,B 11.0992,C 0.2421,E1 11.2492,E2 472.4844} C_DIS
LIN {X 128.2511,Y -56.7344,Z 165,A -22.8338,B 11.0992,C 0.2435,E1 11.2478,E2 473.751} C_DIS
LIN {X 127.0493,Y -59.3768,Z 165,A -24.2041,B 11.0989,C 0.2518,E1 11.2462,E2 475.1465} C_DIS
LIN {X 125.2934,Y -62.9987,Z 165,A -25.8599,B 11.0989,C 0.2565,E1 11.2441,E2 476.8056} C_DIS
LIN {X 123.2735,Y -66.8663,Z 165,A -27.4882,B 11.0989,C 0.257,E1 11.242,E2 478.4161} C_DIS
LIN {X 121.5962,Y -69.8707,Z 165,A -28.8917,B 11.0987,C 0.2606,E1 11.2401,E2 479.8209} C_DIS
LIN {X 119.4171,Y -73.532,Z 165,A -30.6519,B 11.0987,C 0.2656,E1 11.2375,E2 481.5856} C_DIS
LIN {X 117.1139,Y -77.1473,Z 165,A -32.3415,B 11.0986,C 0.2684,E1 11.235,E2 483.2691} C_DIS
LIN {X 115.1335,Y -80.0727,Z 165,A -33.8907,B 11.0984,C 0.2749,E1 11.2325,E2 484.8337} C_DIS
LIN {X 112.6576,Y -83.5207,Z 165,A -35.5203,B 11.0984,C 0.2762,E1 11.2299,E2 486.4517} C_DIS
LIN {X 110.0589,Y -86.9167,Z 165,A -37.2093,B 11.0984,C 0.2788,E1 11.227,E2 488.1351} C_DIS
LIN {X 107.8942,Y -89.5892,Z 165,A -38.6038,B 11.0982,C 0.2818,E1 11.2245,E2 489.5298} C_DIS
LIN {X 105.5977,Y -92.2848,Z 165,A -40.1601,B 11.0981,C 0.2882,E1 11.2216,E2 491.1019} C_DIS
LIN {X 102.782,Y -95.411,Z 165,A -41.721,B 11.0981,C 0.2877,E1 11.2187,E2 492.6442} C_DIS
LIN {X 100.411,Y -97.9037,Z 165,A -43.1187,B 11.0981,C 0.2906,E1 11.216,E2 494.0424} C_DIS
LIN {X 97.9429,Y -100.3727,Z 165,A -44.5298,B 11.0979,C 0.2933,E1 11.2132,E2 495.4532} C_DIS
LIN {X 95.4514,Y -102.7443,Z 165,A -45.9335,B 11.0979,C 0.2962,E1 11.2104,E2 496.8581} C_DIS
LIN {X 92.2893,Y -105.5938,Z 165,A -47.6418,B 11.0978,C 0.2989,E1 11.2068,E2 498.5642} C_DIS
LIN {X 89.3967,Y -108.0537,Z 165,A -49.2704,B 11.0976,C 0.3041,E1 11.2033,E2 500.2045} C_DIS
LIN {X 86.2832,Y -110.5566,Z 165,A -50.8128,B 11.0976,C 0.3048,E1 11.1999,E2 501.7369} C_DIS
LIN {X 82.8885,Y -113.1233,Z 165,A -52.5342,B 11.0976,C 0.3076,E1 11.1961,E2 503.4577} C_DIS
LIN {X 80.0053,Y -115.1804,Z 165,A -54.0952,B 11.0974,C 0.3132,E1 11.1925,E2 505.0349} C_DIS
LIN {X 76.4796,Y -117.551,Z 165,A -55.6787,B 11.0974,C 0.3121,E1 11.1888,E2 506.6004} C_DIS
LIN {X 73.5297,Y -119.4186,Z 165,A -57.2252,B 11.0973,C 0.3177,E1 11.1851,E2 508.1639} C_DIS
LIN {X 69.8719,Y -121.5955,Z 165,A -58.8226,B 11.0973,C 0.3167,E1 11.1813,E2 509.7445} C_DIS
LIN {X 66.8698,Y -123.2716,Z 165,A -60.2849,B 11.0972,C 0.3204,E1 11.1777,E2 511.2156} C_DIS
LIN {X 63.876,Y -124.8468,Z 165,A -61.5997,B 11.0972,C 0.3206,E1 11.1745,E2 512.5229} C_DIS
LIN {X 60.594,Y -126.4721,Z 165,A -63.1791,B 11.0971,C 0.3249,E1 11.1705,E2 514.1144} C_DIS
LIN {X 56.9946,Y -128.1347,Z 165,A -64.7107,B 11.0971,C 0.3248,E1 11.1666,E2 515.6359} C_DIS
LIN {X 53.6616,Y -129.5663,Z 165,A -66.1526,B 11.0971,C 0.3256,E1 11.1629,E2 517.0738} C_DIS
LIN {X 50.4684,Y -130.843,Z 165,A -67.5597,B 11.097,C 0.3273,E1 11.1593,E2 518.4824} C_DIS
LIN {X 47.2452,Y -132.041,Z 165,A -68.9445,B 11.097,C 0.3284,E1 11.1556,E2 519.8657} C_DIS
LIN {X 43.9937,Y -133.1597,Z 165,A -70.3541,B 11.097,C 0.33,E1 11.1519,E2 521.277} C_DIS
LIN {X 40.8123,Y -134.1687,Z 165,A -71.7107,B 11.0969,C 0.3312,E1 11.1483,E2 522.6338} C_DIS
LIN {X 37.5097,Y -135.1294,Z 165,A -73.089,B 11.0969,C 0.3318,E1 11.1446,E2 524.0096} C_DIS
LIN {X 34.075,Y -136.0366,Z 165,A -74.544,B 11.0969,C 0.3331,E1 11.1406,E2 525.4662} C_DIS
LIN {X 30.8141,Y -136.8121,Z 165,A -75.9249,B 11.0968,C 0.3345,E1 11.1369,E2 526.8495} C_DIS
LIN {X 27.3474,Y -137.5478,Z 165,A -77.3557,B 11.0968,C 0.3351,E1 11.133,E2 528.2791} C_DIS
LIN {X 23.9717,Y -138.1767,Z 165,A -78.7494,B 11.0968,C 0.3358,E1 11.1291,E2 529.6726} C_DIS
LIN {X 20.5801,Y -138.7225,Z 165,A -80.1417,B 11.0968,C 0.3363,E1 11.1253,E2 531.0643} C_DIS
LIN {X 17.276,Y -139.1722,Z 165,A -81.5611,B 11.0967,C 0.3385,E1 11.1214,E2 532.4919} C_DIS
LIN {X 13.7661,Y -139.562,Z 165,A -82.9685,B 11.0967,C 0.3382,E1 11.1175,E2 533.8956} C_DIS
LIN {X 10.4417,Y -139.8498,Z 165,A -84.3506,B 11.0967,C 0.3392,E1 11.1136,E2 535.2809} C_DIS
LIN {X 6.9851,Y -140.0648,Z 165,A -85.7319,B 11.0967,C 0.3387,E1 11.1098,E2 536.6585} C_DIS
LIN {X 3.4477,Y -140.1972,Z 165,A -87.1631,B 11.0967,C 0.3387,E1 11.1058,E2 538.0886} C_DIS
LIN {X 0.9957,Y -140.2345,Z 165,A -87.8898,B 11.0969,C 0.332,E1 11.1038,E2 538.7799} C_DIS
Enddeposition()
LIN {X 0.952,Y -131.2651,Z 166,A -88.3469,B 11.338,C 0.2635,E1 11.3429,E2 538.8705} C_DIS
Startdeposition()
$VEL.CP = VEL_PRINT
LIN {X 4.6143,Y -131.1882,Z 166,A -86.2805,B 11.3383,C 0.2521,E1 11.3488,E2 536.7469} C_DIS
LIN {X 7.85,Y -131.0336,Z 166,A -84.9279,B 11.3383,C 0.2531,E1 11.3526,E2 535.401} C_DIS
LIN {X 11.2571,Y -130.7849,Z 166,A -83.4778,B 11.3383,C 0.2535,E1 11.3566,E2 533.955} C_DIS
LIN {X 14.4592,Y -130.4702,Z 166,A -82.0524,B 11.3383,C 0.2524,E1 11.3606,E2 532.5263} C_DIS
LIN {X 17.4527,Y -130.1034,Z 166,A -80.7374,B 11.3383,C 0.2518,E1 11.3642,E2 531.2107} C_DIS
LIN {X 20.6554,Y -129.6342,Z 166,A -79.33,B 11.3383,C 0.2511,E1 11.3681,E2 529.803} C_DIS
LIN {X 23.8266,Y -129.0896,Z 166,A -77.9287,B 11.3383,C 0.2503,E1 11.372,E2 528.4012} C_DIS
LIN {X 27.1811,Y -128.4242,Z 166,A -76.4983,B 11.3383,C 0.2507,E1 11.3759,E2 526.9773} C_DIS
LIN {X 31.1201,Y -127.5264,Z 166,A -74.5844,B 11.3384,C 0.2456,E1 11.3811,E2 525.0439} C_DIS
LIN {X 34.7638,Y -126.5826,Z 166,A -72.9794,B 11.3384,C 0.2451,E1 11.3854,E2 523.4423} C_DIS
LIN {X 37.775,Y -125.7171,Z 166,A -71.7194,B 11.3384,C 0.2464,E1 11.3888,E2 522.1943} C_DIS
LIN {X 41.3556,Y -124.5833,Z 166,A -69.9223,B 11.3385,C 0.2408,E1 11.3936,E2 520.3767} C_DIS
LIN {X 45.7345,Y -123.0436,Z 166,A -68.0938,B 11.3385,C 0.2435,E1 11.3983,E2 518.5706} C_DIS
LIN {X 48.736,Y -121.886,Z 166,A -66.6344,B 11.3385,C 0.2404,E1 11.4022,E2 517.1033} C_DIS
LIN {X 51.7078,Y -120.6554,Z 166,A -65.2399,B 11.3385,C 0.2389,E1 11.4057,E2 515.7087} C_DIS
LIN {X 54.3624,Y -119.4848,Z 166,A -63.9018,B 11.3386,C 0.2354,E1 11.4092,E2 514.3609} C_DIS
LIN {X 57.0647,Y -118.2165,Z 166,A -62.5772,B 11.3386,C 0.233,E1 11.4125,E2 513.0325} C_DIS
LIN {X 60.4598,Y -116.5172,Z 166,A -61.0999,B 11.3386,C 0.2352,E1 11.4162,E2 511.5755} C_DIS
LIN {X 63.2987,Y -115.0007,Z 166,A -59.6471,B 11.3387,C 0.2319,E1 11.4197,E2 510.1157} C_DIS
LIN {X 66.0985,Y -113.4147,Z 166,A -58.3543,B 11.3387,C 0.2325,E1 11.4228,E2 508.8351} C_DIS
LIN {X 68.8585,Y -111.7602,Z 166,A -56.8491,B 11.3387,C 0.2276,E1 11.4265,E2 507.3164} C_DIS
LIN {X 71.4084,Y -110.1482,Z 166,A -55.5434,B 11.3388,C 0.2257,E1 11.4295,E2 506.0107} C_DIS
LIN {X 74.2663,Y -108.2417,Z 166,A -54.0593,B 11.3388,C 0.2234,E1 11.433,E2 504.527} C_DIS
LIN {X 76.7341,Y -106.5072,Z 166,A -52.7059,B 11.3389,C 0.2201,E1 11.4361,E2 503.1678} C_DIS
LIN {X 79.4789,Y -104.4748,Z 166,A -51.1356,B 11.339,C 0.2153,E1 11.4396,E2 501.5863} C_DIS
LIN {X 82.7165,Y -101.9308,Z 166,A -49.3582,B 11.339,C 0.2123,E1 11.4435,E2 499.8096} C_DIS
LIN {X 85.818,Y -99.3331,Z 166,A -47.6037,B 11.3392,C 0.209,E1 11.4472,E2 498.0546} C_DIS
LIN {X 89.2615,Y -96.2508,Z 166,A -45.7246,B 11.3392,C 0.2084,E1 11.451,E2 496.1901} C_DIS
LIN {X 91.662,Y -93.9679,Z 166,A -44.293,B 11.3392,C 0.2057,E1 11.4539,E2 494.7587} C_DIS
LIN {X 94.4472,Y -91.1676,Z 166,A -42.5725,B 11.3392,C 0.202,E1 11.4573,E2 493.0367} C_DIS
LIN {X 97.2606,Y -88.1597,Z 166,A -40.6921,B 11.3394,C 0.1958,E1 11.4609,E2 491.1443} C_DIS
LIN {X 99.9778,Y -85.0659,Z 166,A -38.9183,B 11.3394,C 0.1923,E1 11.4641,E2 489.3714} C_DIS
LIN {X 102.928,Y -81.4722,Z 166,A -37.0209,B 11.3394,C 0.191,E1 11.4674,E2 487.4877} C_DIS
LIN {X 105.3134,Y -78.3636,Z 166,A -35.347,B 11.3395,C 0.1878,E1 11.4702,E2 485.8164} C_DIS
LIN {X 106.9517,Y -76.1129,Z 166,A -34.0578,B 11.3395,C 0.1828,E1 11.4723,E2 484.5167} C_DIS
LIN {X 109.0268,Y -73.1095,Z 166,A -32.5215,B 11.3396,C 0.1804,E1 11.4747,E2 482.9856} C_DIS
LIN {X 110.9035,Y -70.2298,Z 166,A -31.1392,B 11.3396,C 0.1797,E1 11.4768,E2 481.6159} C_DIS
LIN {X 112.489,Y -67.6615,Z 166,A -29.7801,B 11.3397,C 0.1752,E1 11.4788,E2 480.2502} C_DIS
LIN {X 114.455,Y -64.2792,Z 166,A -28.0312,B 11.3398,C 0.1696,E1 11.4812,E2 478.4943} C_DIS
LIN {X 116.5149,Y -60.4642,Z 166,A -26.2312,B 11.3398,C 0.167,E1 11.4836,E2 476.7033} C_DIS
LIN {X 117.8647,Y -57.7862,Z 166,A -24.9096,B 11.3398,C 0.1632,E1 11.4852,E2 475.3787} C_DIS
LIN {X 119.2331,Y -54.9067,Z 166,A -23.5467,B 11.3399,C 0.1602,E1 11.4868,E2 474.0176} C_DIS
LIN {X 120.571,Y -51.9029,Z 166,A -22.1402,B 11.3399,C 0.157,E1 11.4884,E2 472.6129} C_DIS
LIN {X 121.8827,Y -48.7443,Z 166,A -20.5185,B 11.3401,C 0.1494,E1 11.4901,E2 470.9739} C_DIS
LIN {X 123.5272,Y -44.4108,Z 166,A -18.6693,B 11.3401,C 0.1484,E1 11.4919,E2 469.1435} C_DIS
LIN {X 124.5782,Y -41.3709,Z 166,A -17.2809,B 11.3401,C 0.1448,E1 11.4931,E2 467.7553} C_DIS
LIN {X 125.6163,Y -38.1043,Z 166,A -15.8074,B 11.3401,C 0.1412,E1 11.4943,E2 466.2829} C_DIS
LIN {X 126.4574,Y -35.2113,Z 166,A -14.4821,B 11.3402,C 0.1371,E1 11.4954,E2 464.9548} C_DIS
LIN {X 127.3302,Y -31.9134,Z 166,A -13.0634,B 11.3402,C 0.1347,E1 11.4963,E2 463.5429} C_DIS
LIN {X 128.0722,Y -28.7925,Z 166,A -11.6615,B 11.3403,C 0.1306,E1 11.4972,E2 462.1393} C_DIS
LIN {X 128.6961,Y -25.8598,Z 166,A -10.3457,B 11.3403,C 0.1266,E1 11.498,E2 460.8211} C_DIS
LIN {X 129.3386,Y -22.4352,Z 166,A -8.8746,B 11.3403,C 0.1236,E1 11.4987,E2 459.3544} C_DIS
LIN {X 129.8495,Y -19.2594,Z 166,A -7.4648,B 11.3404,C 0.1193,E1 11.4993,E2 457.9423} C_DIS
LIN {X 130.2819,Y -16.0703,Z 166,A -6.1457,B 11.3404,C 0.1174,E1 11.4998,E2 456.632} C_DIS
LIN {X 130.5856,Y -13.3866,Z 166,A -4.7936,B 11.3405,C 0.1094,E1 11.5002,E2 455.2577} C_DIS
LIN {X 130.8975,Y -9.8644,Z 166,A -3.3559,B 11.3405,C 0.1076,E1 11.5005,E2 453.8311} C_DIS
LIN {X 131.1105,Y -6.4366,Z 166,A -1.9623,B 11.3405,C 0.106,E1 11.5007,E2 452.4484} C_DIS
LIN {X 131.2208,Y -3.5371,Z 166,A -0.6678,B 11.3406,C 0.1015,E1 11.5008,E2 451.1493} C_DIS
LIN {X 131.2723,Y -0.0068,Z 166,A 0.8747,B 11.3406,C 0.097,E1 11.5008,E2 449.6051} C_DIS
LIN {X 131.2298,Y 3.213,Z 166,A 2.1899,B 11.3406,C 0.0952,E1 11.5008,E2 448.2992} C_DIS
LIN {X 131.1187,Y 6.2751,Z 166,A 3.5538,B 11.3406,C 0.0906,E1 11.5006,E2 446.9307} C_DIS
LIN {X 130.9272,Y 9.4571,Z 166,A 4.9607,B 11.3407,C 0.0861,E1 11.5004,E2 445.5206} C_DIS
LIN {X 130.6558,Y 12.6664,Z 166,A 6.3341,B 11.3407,C 0.0829,E1 11.5,E2 444.1496} C_DIS
LIN {X 130.2829,Y 16.062,Z 166,A 7.7604,B 11.3407,C 0.0802,E1 11.4995,E2 442.7297} C_DIS
LIN {X 129.8924,Y 18.9595,Z 166,A 9.0451,B 11.3407,C 0.0763,E1 11.499,E2 441.4427} C_DIS
LIN {X 129.371,Y 22.2464,Z 166,A 10.4678,B 11.3408,C 0.0729,E1 11.4984,E2 440.0222} C_DIS
LIN {X 128.7879,Y 25.4087,Z 166,A 11.9361,B 11.3408,C 0.0672,E1 11.4976,E2 438.5448} C_DIS
LIN {X 128.1257,Y 28.5584,Z 166,A 13.3965,B 11.3408,C 0.0617,E1 11.4967,E2 437.0765} C_DIS
LIN {X 127.1185,Y 32.7476,Z 166,A 15.0998,B 11.3408,C 0.061,E1 11.4956,E2 435.3927} C_DIS
LIN {X 126.071,Y 36.5719,Z 166,A 16.7568,B 11.3409,C 0.0581,E1 11.4944,E2 433.743} C_DIS
LIN {X 125.1973,Y 39.4611,Z 166,A 18.1721,B 11.3409,C 0.0518,E1 11.4932,E2 432.3149} C_DIS
LIN {X 124.1281,Y 42.7035,Z 166,A 19.5882,B 11.3409,C 0.0497,E1 11.4919,E2 430.9064} C_DIS
LIN {X 123.0445,Y 45.7322,Z 166,A 20.9102,B 11.3409,C 0.048,E1 11.4907,E2 429.593} C_DIS
LIN {X 121.8872,Y 48.7329,Z 166,A 22.3598,B 11.3409,C 0.043,E1 11.4892,E2 428.1368} C_DIS
LIN {X 120.765,Y 51.4543,Z 166,A 23.7173,B 11.3409,C 0.0376,E1 11.4877,E2 426.7697} C_DIS
LIN {X 119.3455,Y 54.6637,Z 166,A 25.0177,B 11.3409,C 0.0396,E1 11.4862,E2 425.4957} C_DIS
LIN {X 118.0583,Y 57.3938,Z 166,A 26.5123,B 11.341,C 0.0315,E1 11.4844,E2 423.979} C_DIS
LIN {X 116.518,Y 60.4583,Z 166,A 27.864,B 11.341,C 0.0315,E1 11.4827,E2 422.6435} C_DIS
LIN {X 115.0049,Y 63.2909,Z 166,A 29.3058,B 11.341,C 0.0268,E1 11.4808,E2 421.196} C_DIS
LIN {X 113.423,Y 66.0841,Z 166,A 30.7022,B 11.341,C 0.0234,E1 11.4789,E2 419.7993} C_DIS
LIN {X 111.7734,Y 68.8369,Z 166,A 31.9748,B 11.341,C 0.0233,E1 11.477,E2 418.541} C_DIS
LIN {X 110.1428,Y 71.4167,Z 166,A 33.3982,B 11.341,C 0.0177,E1 11.4749,E2 417.1058} C_DIS
LIN {X 108.2458,Y 74.2604,Z 166,A 34.8753,B 11.341,C 0.0145,E1 11.4726,E2 415.6296} C_DIS
LIN {X 106.5009,Y 76.7428,Z 166,A 36.2316,B 11.341,C 0.0105,E1 11.4704,E2 414.2688} C_DIS
LIN {X 104.6572,Y 79.2381,Z 166,A 37.5714,B 11.341,C 0.0078,E1 11.4681,E2 412.9299} C_DIS
LIN {X 102.0564,Y 82.5609,Z 166,A 39.3676,B 11.341,C 0.0048,E1 11.465,E2 411.1381} C_DIS
LIN {X 99.7538,Y 85.3294,Z 166,A 41.0258,B 11.341,C -0.0009,E1 11.462,E2 409.469} C_DIS
LIN {X 97.2598,Y 88.1607,Z 166,A 42.6655,B 11.341,C -0.0043,E1 11.4589,E2 407.8293} C_DIS
LIN {X 94.4434,Y 91.1715,Z 166,A 44.4435,B 11.341,C -0.0075,E1 11.4555,E2 406.0531} C_DIS
LIN {X 91.1712,Y 94.4436,Z 166,A 46.3537,B 11.341,C -0.0088,E1 11.4517,E2 404.1551} C_DIS
LIN {X 88.1603,Y 97.2601,Z 166,A 48.2301,B 11.341,C -0.0142,E1 11.4479,E2 402.269} C_DIS
LIN {X 85.0552,Y 99.9869,Z 166,A 50.0245,B 11.341,C -0.0174,E1 11.4441,E2 400.4751} C_DIS
LIN {X 81.4647,Y 102.9339,Z 166,A 51.9218,B 11.341,C -0.0177,E1 11.44,E2 398.5925} C_DIS
LIN {X 78.3574,Y 105.318,Z 166,A 53.5999,B 11.341,C -0.0199,E1 11.4362,E2 396.9177} C_DIS
LIN {X 75.5929,Y 107.3195,Z 166,A 54.9689,B 11.341,C -0.0194,E1 11.4332,E2 395.5626} C_DIS
LIN {X 73.1119,Y 109.0252,Z 166,A 56.4278,B 11.341,C -0.0251,E1 11.4298,E2 394.0864} C_DIS
LIN {X 70.2526,Y 110.8891,Z 166,A 57.8164,B 11.341,C -0.0249,E1 11.4265,E2 392.7094} C_DIS
Enddeposition()
END
